                        IF fb_json.HasMember(json_FeederConfig, 'InFilterDelay') THEN
                            json_value := fb_json.FindMember(json_FeederConfig, 'InFilterDelay');
                            PERS.recipeList[i + 0].st110.FeederConfig.InFilterDelay
                                := TO_DINT(fb_json.GetInt(json_value));
                        END_IF

                        IF fb_json.HasMember(json_FeederConfig, 'StartDelay') THEN
                            json_value := fb_json.FindMember(json_FeederConfig, 'StartDelay');
                            PERS.recipeList[i + 0].st110.FeederConfig.StartDelay
                                := TO_DINT(fb_json.GetInt(json_value));
                        END_IF

                        IF fb_json.HasMember(json_FeederConfig, 'StopDelay') THEN
                            json_value := fb_json.FindMember(json_FeederConfig, 'StopDelay');
                            PERS.recipeList[i + 0].st110.FeederConfig.StopDelay
                                := TO_DINT(fb_json.GetInt(json_value));
                        END_IF

                        IF fb_json.HasMember(json_FeederConfig, 'EmptyDelay') THEN
                            json_value := fb_json.FindMember(json_FeederConfig, 'EmptyDelay');
                            PERS.recipeList[i + 0].st110.FeederConfig.EmptyDelay
                                := TO_DINT(fb_json.GetInt(json_value));
                        END_IF
                    END_IF
                END_IF

                IF fb_json.HasMember(json_i, 'st115') THEN
                    json_st115 := fb_json.FindMember(json_i, 'st115');

                    IF fb_json.HasMember(json_st115, 'xUseVerLeft') THEN
                        json_value                               := fb_json.FindMember(json_st115, 'xUseVerLeft');
                        PERS.recipeList[i + 0].st115.xUseVerLeft := TO_BOOL(fb_json.GetBool(json_value));
                    END_IF

                    IF fb_json.HasMember(json_st115, 'xUseVerRight') THEN
                        json_value                                := fb_json.FindMember(json_st115, 'xUseVerRight');
                        PERS.recipeList[i + 0].st115.xUseVerRight := TO_BOOL(fb_json.GetBool(json_value));
                    END_IF

                    IF fb_json.HasMember(json_st115, 'FeederConfig') THEN
                        json_FeederConfig := fb_json.FindMember(json_st115, 'FeederConfig');

                        IF fb_json.HasMember(json_FeederConfig, 'InFilterDelay') THEN
                            json_value := fb_json.FindMember(json_FeederConfig, 'InFilterDelay');
                            PERS.recipeList[i + 0].st115.FeederConfig.InFilterDelay
                                := TO_DINT(fb_json.GetInt(json_value));
                        END_IF

                        IF fb_json.HasMember(json_FeederConfig, 'StartDelay') THEN
                            json_value := fb_json.FindMember(json_FeederConfig, 'StartDelay');
                            PERS.recipeList[i + 0].st115.FeederConfig.StartDelay
                                := TO_DINT(fb_json.GetInt(json_value));
                        END_IF

                        IF fb_json.HasMember(json_FeederConfig, 'StopDelay') THEN
                            json_value := fb_json.FindMember(json_FeederConfig, 'StopDelay');
                            PERS.recipeList[i + 0].st115.FeederConfig.StopDelay
                                := TO_DINT(fb_json.GetInt(json_value));
                        END_IF

                        IF fb_json.HasMember(json_FeederConfig, 'EmptyDelay') THEN
                            json_value := fb_json.FindMember(json_FeederConfig, 'EmptyDelay');
                            PERS.recipeList[i + 0].st115.FeederConfig.EmptyDelay
                                := TO_DINT(fb_json.GetInt(json_value));
                        END_IF
                    END_IF
                END_IF

                IF fb_json.HasMember(json_i, 'st120') THEN
                    json_st120 := fb_json.FindMember(json_i, 'st120');

                    IF fb_json.HasMember(json_st120, 'xUseVerLeft') THEN
                        json_value                               := fb_json.FindMember(json_st120, 'xUseVerLeft');
                        PERS.recipeList[i + 0].st120.xUseVerLeft := TO_BOOL(fb_json.GetBool(json_value));
                    END_IF

                    IF fb_json.HasMember(json_st120, 'xUseVerRight') THEN
                        json_value                                := fb_json.FindMember(json_st120, 'xUseVerRight');
                        PERS.recipeList[i + 0].st120.xUseVerRight := TO_BOOL(fb_json.GetBool(json_value));
                    END_IF

                    IF fb_json.HasMember(json_st120, 'FeederConfigLeft') THEN
                        json_FeederConfigLeft := fb_json.FindMember(json_st120, 'FeederConfigLeft');

                        IF fb_json.HasMember(json_FeederConfigLeft, 'InFilterDelay') THEN
                            json_value := fb_json.FindMember(json_FeederConfigLeft, 'InFilterDelay');
                            PERS.recipeList[i + 0].st120.FeederConfigLeft.InFilterDelay
                                := TO_DINT(fb_json.GetInt(json_value));
                        END_IF

                        IF fb_json.HasMember(json_FeederConfigLeft, 'StartDelay') THEN
                            json_value := fb_json.FindMember(json_FeederConfigLeft, 'StartDelay');
                            PERS.recipeList[i + 0].st120.FeederConfigLeft.StartDelay
                                := TO_DINT(fb_json.GetInt(json_value));
                        END_IF

                        IF fb_json.HasMember(json_FeederConfigLeft, 'StopDelay') THEN
                            json_value := fb_json.FindMember(json_FeederConfigLeft, 'StopDelay');
                            PERS.recipeList[i + 0].st120.FeederConfigLeft.StopDelay
                                := TO_DINT(fb_json.GetInt(json_value));
                        END_IF

                        IF fb_json.HasMember(json_FeederConfigLeft, 'EmptyDelay') THEN
                            json_value := fb_json.FindMember(json_FeederConfigLeft, 'EmptyDelay');
                            PERS.recipeList[i + 0].st120.FeederConfigLeft.EmptyDelay
                                := TO_DINT(fb_json.GetInt(json_value));
                        END_IF
                    END_IF

                    IF fb_json.HasMember(json_st120, 'FeederConfigRight') THEN
                        json_FeederConfigRight := fb_json.FindMember(json_st120, 'FeederConfigRight');

                        IF fb_json.HasMember(json_FeederConfigRight, 'InFilterDelay') THEN
                            json_value := fb_json.FindMember(json_FeederConfigRight, 'InFilterDelay');
                            PERS.recipeList[i + 0].st120.FeederConfigRight.InFilterDelay
                                := TO_DINT(fb_json.GetInt(json_value));
                        END_IF

                        IF fb_json.HasMember(json_FeederConfigRight, 'StartDelay') THEN
                            json_value := fb_json.FindMember(json_FeederConfigRight, 'StartDelay');
                            PERS.recipeList[i + 0].st120.FeederConfigRight.StartDelay
                                := TO_DINT(fb_json.GetInt(json_value));
                        END_IF

                        IF fb_json.HasMember(json_FeederConfigRight, 'StopDelay') THEN
                            json_value := fb_json.FindMember(json_FeederConfigRight, 'StopDelay');
                            PERS.recipeList[i + 0].st120.FeederConfigRight.StopDelay
                                := TO_DINT(fb_json.GetInt(json_value));
                        END_IF

                        IF fb_json.HasMember(json_FeederConfigRight, 'EmptyDelay') THEN
                            json_value := fb_json.FindMember(json_FeederConfigRight, 'EmptyDelay');
                            PERS.recipeList[i + 0].st120.FeederConfigRight.EmptyDelay
                                := TO_DINT(fb_json.GetInt(json_value));
                        END_IF
                    END_IF
                END_IF

                IF fb_json.HasMember(json_i, 'st125') THEN
                    json_st125 := fb_json.FindMember(json_i, 'st125');

                    IF fb_json.HasMember(json_st125, 'xUseVerLeft') THEN
                        json_value := fb_json.FindMember(json_st125, 'xUseVerLeft');
                        PERS.recipeList[i + 0].st125.xUseVerLeft
                            := TO_BOOL(fb_json.GetBool(json_value));
                    END_IF

                    IF fb_json.HasMember(json_st125, 'xUseVerRight') THEN
                        json_value := fb_json.FindMember(json_st125, 'xUseVerRight');
                        PERS.recipeList[i + 0].st125.xUseVerRight
                            := TO_BOOL(fb_json.GetBool(json_value));
                    END_IF

                    IF fb_json.HasMember(json_st125, 'FeederConfig') THEN
                        json_FeederConfig := fb_json.FindMember(json_st125, 'FeederConfig');

                        IF fb_json.HasMember(json_FeederConfig, 'InFilterDelay') THEN
                            json_value := fb_json.FindMember(json_FeederConfig, 'InFilterDelay');
                            PERS.recipeList[i + 0].st125.FeederConfig.InFilterDelay
                                := TO_DINT(fb_json.GetInt(json_value));
                        END_IF

                        IF fb_json.HasMember(json_FeederConfig, 'StartDelay') THEN
                            json_value := fb_json.FindMember(json_FeederConfig, 'StartDelay');
                            PERS.recipeList[i + 0].st125.FeederConfig.StartDelay
                                := TO_DINT(fb_json.GetInt(json_value));
                        END_IF

                        IF fb_json.HasMember(json_FeederConfig, 'StopDelay') THEN
                            json_value := fb_json.FindMember(json_FeederConfig, 'StopDelay');
                            PERS.recipeList[i + 0].st125.FeederConfig.StopDelay
                                := TO_DINT(fb_json.GetInt(json_value));
                        END_IF

                        IF fb_json.HasMember(json_FeederConfig, 'EmptyDelay') THEN
                            json_value := fb_json.FindMember(json_FeederConfig, 'EmptyDelay');
                            PERS.recipeList[i + 0].st125.FeederConfig.EmptyDelay
                                := TO_DINT(fb_json.GetInt(json_value));
                        END_IF
                    END_IF
                END_IF

                IF fb_json.HasMember(json_i, 'st145') THEN
                    json_st145 := fb_json.FindMember(json_i, 'st145');

                    IF fb_json.HasMember(json_st145, 'xUseVerLeft') THEN
                        json_value := fb_json.FindMember(json_st145, 'xUseVerLeft');
                        PERS.recipeList[i + 0].st145.xUseVerLeft
                            := TO_BOOL(fb_json.GetBool(json_value));
                    END_IF

                    IF fb_json.HasMember(json_st145, 'xUseVerRight') THEN
                        json_value := fb_json.FindMember(json_st145, 'xUseVerRight');
                        PERS.recipeList[i + 0].st145.xUseVerRight
                            := TO_BOOL(fb_json.GetBool(json_value));
                    END_IF

                    IF fb_json.HasMember(json_st145, 'FeederConfig') THEN
                        json_FeederConfig := fb_json.FindMember(json_st145, 'FeederConfig');

                        IF fb_json.HasMember(json_FeederConfig, 'InFilterDelay') THEN
                            json_value := fb_json.FindMember(json_FeederConfig, 'InFilterDelay');
                            PERS.recipeList[i + 0].st145.FeederConfig.InFilterDelay
                                := TO_DINT(fb_json.GetInt(json_value));
                        END_IF

                        IF fb_json.HasMember(json_FeederConfig, 'StartDelay') THEN
                            json_value := fb_json.FindMember(json_FeederConfig, 'StartDelay');
                            PERS.recipeList[i + 0].st145.FeederConfig.StartDelay
                                := TO_DINT(fb_json.GetInt(json_value));
                        END_IF

                        IF fb_json.HasMember(json_FeederConfig, 'StopDelay') THEN
                            json_value := fb_json.FindMember(json_FeederConfig, 'StopDelay');
                            PERS.recipeList[i + 0].st145.FeederConfig.StopDelay
                                := TO_DINT(fb_json.GetInt(json_value));
                        END_IF

                        IF fb_json.HasMember(json_FeederConfig, 'EmptyDelay') THEN
                            json_value := fb_json.FindMember(json_FeederConfig, 'EmptyDelay');
                            PERS.recipeList[i + 0].st145.FeederConfig.EmptyDelay
                                := TO_DINT(fb_json.GetInt(json_value));
                        END_IF
                    END_IF
                END_IF
            END_IF

            IF fb_json.HasMember(json_i, 'st180') THEN
                json_st180 := fb_json.FindMember(json_i, 'st180');

                IF fb_json.HasMember(json_st180, 'xUseVerLeft') THEN
                    json_value                               := fb_json.FindMember(json_st180, 'xUseVerLeft');
                    PERS.recipeList[i + 0].st180.xUseVerLeft := TO_BOOL(fb_json.GetBool(json_value));
                END_IF

                IF fb_json.HasMember(json_st180, 'xUseVerRight') THEN
                    json_value                                := fb_json.FindMember(json_st180, 'xUseVerRight');
                    PERS.recipeList[i + 0].st180.xUseVerRight := TO_BOOL(fb_json.GetBool(json_value));
                END_IF
            END_IF
        END_FOR
    END_IF
END_IF

IF fb_json.HasMember(json_head, 'iRecipeCurrent') THEN
    json_value          := fb_json.FindMember(json_head, 'iRecipeCurrent');
    PERS.iRecipeCurrent := TO_INT(fb_json.GetInt(json_value));
END_IF

END_FUNCTION

// ---- POUs/20_AUTO/FileMan/LoadFromMemory.TcPOU
FUNCTION LoadFromMemory : BOOL
VAR_INPUT
    sData : REFERENCE TO STRING(2000);
END_VAR
VAR
    fbJson     : FB_JsonSaxReader;
    pJsonParse : FB_ReadJSON;
    //pJsonParse : FB_ReadRecipeJson;

    i : int;
END_VAR

// pJsonParse.myArrayInput1 REF= PERS.iStationTimeDef1;
// pJsonParse.myArrayInput2 REF= PERS.iStationTimeDef2;
fbJson.Parse(sJson := sData, ipHdl := pJsonParse);

END_FUNCTION

// ---- POUs/20_AUTO/FileMan/SaveInMemory.TcPOU
FUNCTION SaveInMemory : BOOL
VAR_INPUT
    sData : REFERENCE TO STRING(2000);
END_VAR
VAR
    fbJson     : FB_JsonSaxWriter;
    i          : int;
END_VAR

fbJson.ResetDocument();
// global object
fbJson.StartObject();
fbJson.AddKey('StationTimeArray');

// array1
fbJson.StartObject();
fbJson.AddKey('StationTime1');
fbJson.StartArray();

FOR i := 1 TO CONST.STATION_NUMBER BY 1 DO
    fbJson.AddDint(PERS.iStationTimeDef1[i]);
END_FOR

fbJson.EndArray();

// array2
fbJson.AddKey('StationTime2');
fbJson.StartArray();

FOR i := 1 TO CONST.STATION_NUMBER BY 1 DO
    fbJson.AddDint(PERS.iStationTimeDef2[i]);
END_FOR


fbJson.EndArray();
fbJson.EndObject();

fbJson.EndObject();
// end global object

// end of file
sData := fbJson.GetDocument();

fbJson.ResetDocument();

END_FUNCTION

// ---- POUs/20_AUTO/ST100/FB_ABL_LASER.TcPOU
FUNCTION_BLOCK FB_ABL_LASER
(****************************************************************************************)
(*	TITEL				Bezeichnung Ablauf	    										*)
(*	Status				ungetestet                         								*)
(*  Version:			1.0																*)
(*	Beschrieb:			Ablaufbeschreibung												*)
(*																						*)
(*	Steps:																				*)
(*		RESET:=0		Reset der Station												*)
(* 		INIT:=100		Initialisieren													*)
(*		... 			...																*)
(*		READY:=999		Initialisiert, Bereit für Start									*)
(*		START:=1000		Start Zyklisch 													*)
(*		... 			...																*)
(*		DONE:=8000		Letzer Schritt													*)
(*		ERROR:=9000		ALARM/Fehler													*)
(* 	09.09.2019/Dj																		*)
(***********************************Revisionen*******************************************)
(*	dd.mm.yyyy   KZ    x.y			Beschrieb											*)
(****************************************************************************************)

VAR_INPUT
    xIN_Reset       : BOOL;          // Schrittkette zurücksetzen 
    xIN_Init        : BOOL;          // Initialisieren
    xIN_Quit        : BOOL;          // Fehler quittieren 
    xIN_Start       : BOOL;          // Startbefehl
    xIN_Sperre      : BOOL;          // FB Sperren 
    xIN_NextStep    : BOOL;          // Nächsten Schritt ausführen 
    xIN_AlarmAktiv  : BOOL;          // Anlage hat Alarm
    xIN_DryCycle    : BOOL;          // Fahren ohne Teile
    xIN_RestartCYCL : BOOL;          // Zyklus erneut starten im STEP, END, LEERFAHREN
    enIN_State      : enState;       // Status Anlage
    tIN_Timeout     : TIME := T#10s; // Timout

    pxFG_Freigabe : POINTER TO BOOL; //Freigabe von Station

    // Application specific
    iProcessTimeMili1 : UDINT := 5000; // user defined station duration, in milisecond
    iProcessTimeMili2 : UDINT := 5000; // user defined station duration, in milisecond
    Mover            : REFERENCE TO FB_Mover;
    //xIN_MoverInPos  : BOOL;          // Set this flag when a mover is in position and ready to be handled
END_VAR
VAR_OUTPUT
    (* standart Ausgänge *)
    xOUT_ErrFlag     : BOOL;   // Error Flag 
    xOUT_Busy        : BOOL;   // Baustein befindet sich im Ablauf 
    xOUT_Done        : BOOL;   // Baustein hat den Ablauf beendet 		
    xOUT_Ready       : BOOL;   // Ready to begin, should be the same state as done	
    xOUT_Timeout     : BOOL;   // Timeout FB 
    xOUT_InitDone    : BOOL;   // initialisierung fertig
    xOUT_Wait        : BOOL;   // Wartet auf Bedingung
    iOUT_Step        : INT;    // Aktueller Schritt 
    sOUT_Step        : STRING; // Aktueller Schritt but in string format
    bOUT_Error       : BYTE;   // Fehlernummer

    xOUT_MoverFree   : BOOL;   // The mover is free to move
    //xOUT_MoverNeeded : BOOL;   // A mover is needed by this station to continue its process
    iOUT_ProcessCompletion : INT; //process completion, express in % (0-100)
END_VAR
VAR
    (* Standard *)
    (* Schritt *)
    iLastStep : INT; // Merker letzter Schritt 
    iPreStep  : INT; // Schritt zurück nach Alarm 
    iAktStep  : INT; // aktueller Schritt

    // Trigger Starten 
    rtSTART : R_TRIG;
    // Timer TimeOut 
    TON_Timeout : TON;

    (* Bausteine *)

    (* Spezial *)
    iStartProcessTimeMili : UDINT; // start of the processing time, accurate at 100ns 
	
	_bBewegung : BOOL;
	_bBewegungDist : INT := 20;

END_VAR
VAR CONSTANT
END_VAR

(*******************************************************************)
(* Trigger  *)
(*******************************************************************)
(* Zurücksetzen *)
IF xIN_RESET THEN
    iPreStep  := ST100_Laser_e.RESET;
    iOUT_Step := ST100_Laser_e.RESET;
END_IF;

(* Error Quittieren *)
IF (bOUT_Error <> 0) AND xIN_Quit THEN
    xOUT_ErrFlag := FALSE;
    bOUT_Error   := 0;
    iOUT_Step    := iPreStep;
END_IF;

(*******************************************************************)
(* Timer *)
(*******************************************************************)
TON_Timeout(IN := xIN_NextStep AND (iLastStep = iOUT_Step) (*todo FG *) ,
            PT := tIN_Timeout);

(*******************************************************************)
(* Bausteine *)
(*******************************************************************)

(*******************************************************************)
(* OUTPUTS *)
(*******************************************************************)
// Error Flag 
xOUT_ErrFlag := (bOUT_Error <> 0);
// Baustein befindet sich im Ablauf 
xOUT_Busy := (iOUT_Step > ST100_Laser_e.READY) AND (iOUT_Step < ST100_Laser_e.DONE);
// Baustein hat den Ablauf beendet
xOUT_Done := (iOUT_Step = ST100_Laser_e.DONE);
// Process ready
xOUT_Ready := (iOUT_Step = ST100_Laser_e.READY);
// Timeout FB 				 		
xOUT_Timeout := TON_Timeout.Q;
// Itialisierung fertig			
xOUT_InitDone := (iOUT_Step = ST100_Laser_e.READY);
// Aktueller Schritt			
iOUT_Step := iOUT_Step; //Im Ablauf gesetzt		
sOUT_Step := TO_STRING(iOUT_Step);
//Fehlernummer	 
bOUT_Error := bOUT_Error; //Im Ablauf/FB gesetzt	
(* Warte (alle Schritte wo auf FG oder Teile gewartet wird) *)
xOUT_Wait := (iOUT_Step = ST100_Laser_e.DONE);

xOUT_MoverFree := iOUT_Step = ST100_Laser_e.waitOnMover;

iOUT_ProcessCompletion := F_GetPercent(iAktStep,
                                       ST100_Laser_e.START,
                                       ST100_Laser_e.DONE,
                                       ST100_Laser_e.proceedOperation_1,
                                       ST100_Laser_e.proceedOperation_2,
                                       iStartProcessTimeMili,
                                       TO_DINT(iProcessTimeMili1),
                                       TO_DINT(iProcessTimeMili2));

(*******************************************************************)
(* Ablauf *)
(*******************************************************************)

(* Sperren *)
IF xIN_Sperre THEN
    iPreStep  := ST100_Laser_e.RESET;
    iOUT_Step := ST100_Laser_e.RESET;
    RETURN;
END_IF;

(* Schritt Merker *)
IF iAktStep <> iOUT_Step THEN
    iLastStep := iAktStep;
    iAktStep  := iOUT_Step;
END_IF

(* START *)
rtSTART(CLK := xIN_Start);

(*******************************************************************)
(* Schrittkette  *)
(*******************************************************************)
CASE iOUT_Step OF

(***** RESET *****)
ST100_Laser_e.RESET: (* Schritt 0-99 *)
    //Initialisierungen
    //Start Init Ablauf
    IF xIN_Init THEN
        iOUT_Step := ST100_Laser_e.INIT;
        //Start Manu Ablauf
    ELSIF enIN_State = StateMANU AND xIN_NextStep THEN
        iOUT_Step := ST100_Laser_e.INIT;
    END_IF;

(***** INIT *****)
ST100_Laser_e.INIT: (* Grundstellung ? *)
    IF TRUE THEN
        iOUT_Step := ST100_Laser_e.READY;
    ELSE
        iOUT_Step := ST100_Laser_e.INIT;
    END_IF;

(***** READY / INIT DONE *****)
ST100_Laser_e.READY:  (* Start AUTO,END,LEER,STEP *)
    IF xIN_Start THEN //IF rtSTART.Q THEN
        iOUT_Step := ST100_Laser_e.START;
    END_IF

(***** START  ZYKLISCH *****)
ST100_Laser_e.START: (*  *)
    IF xIN_NextStep AND pxFG_Freigabe^ THEN
        iOUT_Step             := ST100_Laser_e.waitOnMover;
        iStartProcessTimeMili := GetTick();
    END_IF;

ST100_Laser_e.waitOnMover: (*  *)
    IF xIN_NextStep AND __ISVALIDREF(Mover) THEN
        iStartProcessTimeMili := GetTick();
        iOUT_Step             := ST100_Laser_e.proceedOperation_1;
    END_IF;

ST100_Laser_e.proceedOperation_1: (*  *)
    IF xIN_NextStep AND (GetTick() - iStartProcessTimeMili) >= (iProcessTimeMili1) THEN
        iStartProcessTimeMili := GetTick();
        iOUT_Step             := ST100_Laser_e.proceedOperation_2;
        _bBewegung            := FALSE;
    END_IF

ST100_Laser_e.move_mover_to_next_piece:
    IF __ISVALIDREF(Mover) THEN
        IF Mover.MoverAxis.RelMoveTo(120.0).isInPos THEN
            iOUT_Step := ST100_Laser_e.proceedOperation_2;
        END_IF
    END_IF;

ST100_Laser_e.proceedOperation_2: (*  *)
    IF xIN_NextStep AND (GetTick() - iStartProcessTimeMili) >= (iProcessTimeMili2) THEN
        iOUT_Step := ST100_Laser_e.SYNC_MOVER_LEAVE;
    END_IF;

ST100_Laser_e.SYNC_MOVER_LEAVE:
    // The mover needs to be taken by MoverMan
    IF NOT __ISVALIDREF(Mover) THEN
        iOUT_Step := ST100_Unload_e.DONE;
    END_IF

(***** DONE *****)
ST100_Laser_e.DONE: (* Letzter Schritt  *)
    IF NOT xIN_AlarmAktiv THEN
        //AUTO
        IF (enIN_State = StateAUTO) AND xIN_RestartCYCL THEN
            iOUT_Step := ST100_Laser_e.START;
            //STEP / END / LEERFAHREN restart
        ELSIF (enIN_State < StateAUTO) AND (enIN_State >= enState.StateSTEP) AND xIN_RestartCYCL THEN
            iOUT_Step := ST100_Laser_e.START;
            //STEP / END / LEERFAHREN fertig
        ELSIF (enIN_State = StateREADY) THEN
            iOUT_Step := ST100_Laser_e.READY;
        END_IF;
    END_IF;

(************ ERROR *************)
ST100_Laser_e.ERROR: (* ERROR *) ;

END_CASE;

END_FUNCTION_BLOCK

// ---- POUs/20_AUTO/ST100/FB_AUT_LASER.TcPOU
FUNCTION_BLOCK FB_AUT_LASER EXTENDS FB_AUT_ABSTRACT IMPLEMENTS ISimuMoverTimers
    (****************************************************************************)
    (*	POU_AUT_zxx			Bausteinaufrufe Station	zxx							*)
    (*	Status				ungetestet											*)
    (*  Version:			1.0													*)
    (*	Beschrieb:																*)
    (*																			*)
    (*	Abläufe:			FB_ABLzxxA		Hauptablauf							*)
    (*																			*)
    (*																			*)
    (* 	25.09.2019/Dj															*)
    (****************************************************************************)
    (*	dd.mm.yyyy   KZ    x.y			Beschrieb								*)
    (****************************************************************************)
VAR_INPUT
    (* spezifische Eingänge *)

END_VAR
VAR_OUTPUT
    (* spezifische Ausgänge *)

END_VAR
VAR
    (* Bausteine *)
    _FB_ABL_100A : FB_ABL_LASER;
END_VAR

(*******************************************************************)
(* Timer *)
(*******************************************************************)

(*******************************************************************)
(* Flanken / Merker *)
(*******************************************************************)
//MANU CYCLE
IF (enIN_State = StateMANU) AND xIN_ManuCycle THEN
    xManuCycle := TRUE;
END_IF;

IF (enIN_State <> StateMANU) OR xOUT_Done THEN
    xManuCycle := FALSE;
END_IF

//NEXT STEP
xNextStep := (enIN_State > StateSTEP) OR
             ((enIN_State = StateSTEP) AND xIN_Step) OR
             ((enIN_State = StateMANU) AND xManuCycle);

//RESET
xReset := (enIN_State < StateREADY) AND (enIN_State <> StateINIT) AND NOT xManuCycle;

(*******************************************************************)
(* Bausteinaufrufe Abläufe *)
(*******************************************************************)

_FB_ABL_100A(xIN_Reset    := xReset,
             xIN_Init     := xIN_Init,
             xIN_Quit     := xIN_Quit,
             xIN_Start    := enIN_State = enState.StateAUTO, //AND _FB_ABL_100A.xOUT_Done AND _FB_ABL_100A.xOUT_Ready,
             xIN_Sperre   := NOT xIN_On,
             xIN_NextStep := xNextStep,
             xIN_AlarmAktiv
                 := xIN_AlarmAktiv,
             xIN_DryCycle    := xIN_DryCycle,
             xIN_RestartCYCL := enIN_State = enState.StateAUTO, // only restart when the mover has move out
             enIN_State      := enIN_State,
             tIN_Timeout     := tIN_Timeout,
             pxFG_Freigabe   := ADR(xRelease),
             Mover           := THIS^.Mover,
             xOUT_ErrFlag    =>,
             xOUT_Busy       =>,
             xOUT_Done       =>,
             xOUT_Timeout    =>,
             xOUT_InitDone   =>,
             xOUT_Wait       =>,
             iOUT_Step       =>,
             bOUT_Error      =>);

(*******************************************************************)
(* Mover reset flags *)
(*******************************************************************)

(*******************************************************************)
(* OUTPUT *)
(*******************************************************************)
xOUT_InitDone := _FB_ABL_100A.xOUT_InitDone;
xOUT_Ready    := xOUT_InitDone;
xOUT_Done     := _FB_ABL_100A.xOUT_Done;
xOUT_ErrFlag  := _FB_ABL_100A.xOUT_ErrFlag;
xOUT_Wait     := _FB_ABL_100A.xOUT_Wait;
xOUT_AlarmST  := xOUT_ErrFlag;

(*******************************************************************)
(* Bausteinaufruf Error Station *)
(*******************************************************************)
// POU_ERR_VORLAGE(xIN_QUIT:=xIN_Quit , pstrArIN_ALARM:=ADR(HMI.strArALARM[1]));

METHOD GiveMover : IProcessSampleMover
VAR_INPUT
	mover : REFERENCE TO FB_Mover;
END_VAR
IF __ISVALIDREF(mover) THEN
    THIS^.Mover                       REF= mover;
END_IF
END_METHOD

(* % of completion of the process *)
PROPERTY iCompletionPC : INT
GET
iCompletionPC := THIS^._FB_ABL_100A.iOUT_ProcessCompletion;
END_GET
END_PROPERTY

(* Process time, expressed in milisecond *)
PROPERTY iProcessTimeMili_1 : DINT
GET
iProcessTimeMili_1 := TO_DINT(this^._FB_ABL_100A.iProcessTimeMili1);
END_GET
SET
THIS^._FB_ABL_100A.iProcessTimeMili1 := TO_UDINT(iProcessTimeMili_1);
END_SET
END_PROPERTY

(* Process time, expressed in milisecond *)
PROPERTY iProcessTimeMili_2 : DINT
GET
iProcessTimeMili_2 := TO_DINT(this^._FB_ABL_100A.iProcessTimeMili2);
END_GET
SET
THIS^._FB_ABL_100A.iProcessTimeMili2 := TO_UDINT(iProcessTimeMili_2);
END_SET
END_PROPERTY

PROPERTY ProcessExecution : ProcessExecution_e
GET
ProcessExecution := THIS^._ProcessExecution;
END_GET
SET
THIS^._ProcessExecution := ProcessExecution;
END_SET
END_PROPERTY

METHOD TakeMover : IProcessSampleMover
VAR_INPUT
END_VAR
THIS^.Mover REF= 0;
END_METHOD

PROPERTY xBusy : BOOL
GET
xBusy := This^._FB_ABL_100A.xOUT_Busy;
END_GET
SET
END_SET
END_PROPERTY

PROPERTY xDone : BOOL
GET
xDone := THIS^._FB_ABL_100A.xOUT_Ready OR THIS^._FB_ABL_100A.xOUT_Done;
END_GET
END_PROPERTY

PROPERTY xMoverPathFree : BOOL
GET
xMoverPathFree := THIS^._FB_ABL_100A.xOUT_MoverFree OR THIS^._FB_ABL_100A.xOUT_Ready OR THIS^._FB_ABL_100A.xOUT_Done;
END_GET
END_PROPERTY

PROPERTY xMoverShouldLeave : BOOL
GET
xMoverShouldLeave := THIS^._FB_ABL_100A.iOUT_Step = ST100_Modify_e.SYNC_MOVER_LEAVE;
END_GET
END_PROPERTY

END_FUNCTION_BLOCK

// ---- POUs/20_AUTO/ST100/FB_AUT_100.TcPOU
FUNCTION_BLOCK FB_AUT_100 EXTENDS FB_AUT_ABSTRACT IMPLEMENTS ISimuMoverTimers
    (****************************************************************************)
    (*	POU_AUT_zxx			Bausteinaufrufe Station	zxx							*)
    (*	Status				ungetestet											*)
    (*  Version:			1.0													*)
    (*	Beschrieb:																*)
    (*																			*)
    (*	Abläufe:			FB_ABLzxxA		Hauptablauf							*)
    (*																			*)
    (*																			*)
    (* 	25.09.2019/Dj															*)
    (****************************************************************************)
    (*	dd.mm.yyyy   KZ    x.y			Beschrieb								*)
    (****************************************************************************)
VAR_INPUT
    (* spezifische Eingänge *)

END_VAR
VAR_OUTPUT
    (* spezifische Ausgänge *)

END_VAR
VAR
    (* Bausteine *)
    _FB_ABL_100A : FB_ABL_LOAD;
END_VAR

(*******************************************************************)
(* Timer *)
(*******************************************************************)

(*******************************************************************)
(* Flanken / Merker *)
(*******************************************************************)
//MANU CYCLE
IF (enIN_State = StateMANU) AND xIN_ManuCycle THEN
    xManuCycle := TRUE;
END_IF;

IF (enIN_State <> StateMANU) OR xOUT_Done THEN
    xManuCycle := FALSE;
END_IF

//NEXT STEP
xNextStep := (enIN_State > StateSTEP) OR
             ((enIN_State = StateSTEP) AND xIN_Step) OR
             ((enIN_State = StateMANU) AND xManuCycle);

//RESET
xReset := (enIN_State < StateREADY) AND (enIN_State <> StateINIT) AND NOT xManuCycle;

(*******************************************************************)
(* Bausteinaufrufe Abläufe *)
(*******************************************************************)

_FB_ABL_100A(xIN_Reset    := xReset,
             xIN_Init     := xIN_Init,
             xIN_Quit     := xIN_Quit,
             xIN_Start    := enIN_State = enState.StateAUTO, //AND _FB_ABL_100A.xOUT_Done AND _FB_ABL_100A.xOUT_Ready,
             xIN_Sperre   := NOT xIN_On,
             xIN_NextStep := xNextStep,
             xIN_AlarmAktiv
                 := xIN_AlarmAktiv,
             xIN_DryCycle    := xIN_DryCycle,
             xIN_RestartCYCL := enIN_State = enState.StateAUTO, // only restart when the mover has move out
             enIN_State      := enIN_State,
             tIN_Timeout     := tIN_Timeout,
             pxFG_Freigabe   := ADR(xRelease),
             Mover           := THIS^.Mover,
             xOUT_ErrFlag    =>,
             xOUT_Busy       =>,
             xOUT_Done       =>,
             xOUT_Timeout    =>,
             xOUT_InitDone   =>,
             xOUT_Wait       =>,
             iOUT_Step       =>,
             bOUT_Error      =>);

(*******************************************************************)
(* Mover reset flags *)
(*******************************************************************)

(*******************************************************************)
(* OUTPUT *)
(*******************************************************************)
xOUT_InitDone := _FB_ABL_100A.xOUT_InitDone;
xOUT_Ready    := xOUT_InitDone;
xOUT_Done     := _FB_ABL_100A.xOUT_Done;
xOUT_ErrFlag  := _FB_ABL_100A.xOUT_ErrFlag;
xOUT_Wait     := _FB_ABL_100A.xOUT_Wait;
xOUT_AlarmST  := xOUT_ErrFlag;

(*******************************************************************)
(* Bausteinaufruf Error Station *)
(*******************************************************************)
// POU_ERR_VORLAGE(xIN_QUIT:=xIN_Quit , pstrArIN_ALARM:=ADR(HMI.strArALARM[1]));

METHOD GiveMover : IProcessSampleMover
VAR_INPUT
	mover : REFERENCE TO FB_Mover;
END_VAR
IF __ISVALIDREF(mover) THEN
    THIS^.Mover                       REF= mover;
END_IF
END_METHOD

(* % of completion of the process *)
PROPERTY iCompletionPC : INT
GET
iCompletionPC := THIS^._FB_ABL_100A.iOUT_ProcessCompletion;
END_GET
END_PROPERTY

(* Process time, expressed in milisecond *)
PROPERTY iProcessTimeMili_1 : DINT
GET
iProcessTimeMili_1 := TO_DINT(this^._FB_ABL_100A.iProcessTimeMili1);
END_GET
SET
THIS^._FB_ABL_100A.iProcessTimeMili1 := TO_UDINT(iProcessTimeMili_1);
END_SET
END_PROPERTY

(* Process time, expressed in milisecond *)
PROPERTY iProcessTimeMili_2 : DINT
GET
iProcessTimeMili_2 := TO_DINT(this^._FB_ABL_100A.iProcessTimeMili2);
END_GET
SET
THIS^._FB_ABL_100A.iProcessTimeMili2 := TO_UDINT(iProcessTimeMili_2);
END_SET
END_PROPERTY

PROPERTY ProcessExecution : ProcessExecution_e
GET
ProcessExecution := THIS^._ProcessExecution;
END_GET
SET
THIS^._ProcessExecution := ProcessExecution;
END_SET
END_PROPERTY

METHOD TakeMover : IProcessSampleMover
VAR_INPUT
END_VAR
THIS^.Mover REF= 0;
END_METHOD

PROPERTY xBusy : BOOL
GET
xBusy := This^._FB_ABL_100A.xOUT_Busy;
END_GET
SET
END_SET
END_PROPERTY

PROPERTY xDone : BOOL
GET
xDone := THIS^._FB_ABL_100A.xOUT_Ready OR THIS^._FB_ABL_100A.xOUT_Done;
END_GET
END_PROPERTY

PROPERTY xMoverPathFree : BOOL
GET
xMoverPathFree := THIS^._FB_ABL_100A.xOUT_MoverFree OR THIS^._FB_ABL_100A.xOUT_Ready OR THIS^._FB_ABL_100A.xOUT_Done;
END_GET
END_PROPERTY

PROPERTY xMoverShouldLeave : BOOL
GET
xMoverShouldLeave := THIS^._FB_ABL_100A.iOUT_Step = ST100_Load_e.SYNC_MOVER_LEAVE;
END_GET
END_PROPERTY

END_FUNCTION_BLOCK

// ---- POUs/20_AUTO/ST100/FB_ABL_LOAD.TcPOU
FUNCTION_BLOCK FB_ABL_LOAD
(****************************************************************************************)
(*	TITEL				Bezeichnung Ablauf	    										*)
(*	Status				ungetestet                         								*)
(*  Version:			1.0																*)
(*	Beschrieb:			Ablaufbeschreibung												*)
(*																						*)
(*	Steps:																				*)
(*		RESET:=0		Reset der Station												*)
(* 		INIT:=100		Initialisieren													*)
(*		... 			...																*)
(*		READY:=999		Initialisiert, Bereit für Start									*)
(*		START:=1000		Start Zyklisch 													*)
(*		... 			...																*)
(*		DONE:=8000		Letzer Schritt													*)
(*		ERROR:=9000		ALARM/Fehler													*)
(* 	09.09.2019/Dj																		*)
(***********************************Revisionen*******************************************)
(*	dd.mm.yyyy   KZ    x.y			Beschrieb											*)
(****************************************************************************************)

VAR_INPUT
    xIN_Reset       : BOOL;          // Schrittkette zurücksetzen 
    xIN_Init        : BOOL;          // Initialisieren
    xIN_Quit        : BOOL;          // Fehler quittieren 
    xIN_Start       : BOOL;          // Startbefehl
    xIN_Sperre      : BOOL;          // FB Sperren 
    xIN_NextStep    : BOOL;          // Nächsten Schritt ausführen 
    xIN_AlarmAktiv  : BOOL;          // Anlage hat Alarm
    xIN_DryCycle    : BOOL;          // Fahren ohne Teile
    xIN_RestartCYCL : BOOL;          // Zyklus erneut starten im STEP, END, LEERFAHREN
    enIN_State      : enState;       // Status Anlage
    tIN_Timeout     : TIME := T#10s; // Timout

    pxFG_Freigabe : POINTER TO BOOL; //Freigabe von Station

    // Application specific
    iProcessTimeMili1 : UDINT := 5000; // user defined station duration, in milisecond
    iProcessTimeMili2 : UDINT := 5000; // user defined station duration, in milisecond
    Mover            : REFERENCE TO FB_Mover;
    //xIN_MoverInPos  : BOOL;          // Set this flag when a mover is in position and ready to be handled
END_VAR
VAR_OUTPUT
    (* standart Ausgänge *)
    xOUT_ErrFlag     : BOOL;   // Error Flag 
    xOUT_Busy        : BOOL;   // Baustein befindet sich im Ablauf 
    xOUT_Done        : BOOL;   // Baustein hat den Ablauf beendet 		
    xOUT_Ready       : BOOL;   // Ready to begin, should be the same state as done	
    xOUT_Timeout     : BOOL;   // Timeout FB 
    xOUT_InitDone    : BOOL;   // initialisierung fertig
    xOUT_Wait        : BOOL;   // Wartet auf Bedingung
    iOUT_Step        : INT;    // Aktueller Schritt 
    sOUT_Step        : STRING; // Aktueller Schritt but in string format
    bOUT_Error       : BYTE;   // Fehlernummer

    iOUT_ProcessCompletion : INT; //process completion, express in % (0-100)
    xOUT_MoverFree   : BOOL;   // The mover is free to move
    //xOUT_MoverNeeded : BOOL;   // A mover is needed by this station to continue its process
END_VAR
VAR
    (* Standard *)
    (* Schritt *)
    iLastStep : INT; // Merker letzter Schritt 
    iPreStep  : INT; // Schritt zurück nach Alarm 
    iAktStep  : INT; // aktueller Schritt

    // Trigger Starten 
    rtSTART : R_TRIG;
    // Timer TimeOut 
    TON_Timeout : TON;

    (* Bausteine *)

    (* Spezial *)
    iStartProcessTimeMili : UDINT; // start of the processing time, accurate at 100ns 

END_VAR
VAR CONSTANT
END_VAR

(*******************************************************************)
(* Trigger  *)
(*******************************************************************)
(* Zurücksetzen *)
IF xIN_RESET THEN
    iPreStep  := ST100_Load_e.RESET;
    iOUT_Step := ST100_Load_e.RESET;
END_IF;

(* Error Quittieren *)
IF (bOUT_Error <> 0) AND xIN_Quit THEN
    xOUT_ErrFlag := FALSE;
    bOUT_Error   := 0;
    iOUT_Step    := iPreStep;
END_IF;

(*******************************************************************)
(* Timer *)
(*******************************************************************)
TON_Timeout(IN := xIN_NextStep AND (iLastStep = iOUT_Step) (*todo FG *) ,
            PT := tIN_Timeout);

(*******************************************************************)
(* Bausteine *)
(*******************************************************************)

(*******************************************************************)
(* OUTPUTS *)
(*******************************************************************)
// Error Flag 
xOUT_ErrFlag := (bOUT_Error <> 0);
// Baustein befindet sich im Ablauf 
xOUT_Busy := (iOUT_Step > ST100_Load_e.READY) AND (iOUT_Step < ST100_Load_e.DONE);
// Baustein hat den Ablauf beendet
xOUT_Done := (iOUT_Step = ST100_Load_e.DONE);
// Process ready
xOUT_Ready := (iOUT_Step = ST100_Load_e.READY);
// Timeout FB 				 		
xOUT_Timeout := TON_Timeout.Q;
// Itialisierung fertig			
xOUT_InitDone := (iOUT_Step = ST100_Load_e.READY);
// Aktueller Schritt			
iOUT_Step := iOUT_Step; //Im Ablauf gesetzt		
sOUT_Step := TO_STRING(iOUT_Step);
//Fehlernummer	 
bOUT_Error := bOUT_Error; //Im Ablauf/FB gesetzt	
(* Warte (alle Schritte wo auf FG oder Teile gewartet wird) *)
xOUT_Wait := (iOUT_Step = ST100_Load_e.DONE);

xOUT_MoverFree := iOUT_Step >= ST100_Load_e.MOVER_FREE_OP AND iOUT_Step < ST100_Load_e.MOVER_NEEDED_OP;

iOUT_ProcessCompletion := F_GetPercent(iAktStep,
                                       ST100_Load_e.START,
                                       ST100_Load_e.DONE,
                                       ST100_Load_e.proceedOperation_1,
                                       ST100_Load_e.proceedOperation_2,
                                       iStartProcessTimeMili,
                                       TO_DINT(iProcessTimeMili1),
                                       TO_DINT(iProcessTimeMili2));

(*******************************************************************)
(* Ablauf *)
(*******************************************************************)

(* Sperren *)
IF xIN_Sperre THEN
    iPreStep  := ST100_Load_e.RESET;
    iOUT_Step := ST100_Load_e.RESET;
    RETURN;
END_IF;

(* Schritt Merker *)
IF iAktStep <> iOUT_Step THEN
    iLastStep := iAktStep;
    iAktStep  := iOUT_Step;
END_IF

(* START *)
rtSTART(CLK := xIN_Start);

(*******************************************************************)
(* Schrittkette  *)
(*******************************************************************)
CASE iOUT_Step OF

(***** RESET *****)
ST100_Load_e.RESET: (* Schritt 0-99 *)
    //Initialisierungen
    //Start Init Ablauf
    IF xIN_Init THEN
        iOUT_Step := ST100_Load_e.INIT;
        //Start Manu Ablauf
    ELSIF enIN_State = StateMANU AND xIN_NextStep THEN
        iOUT_Step := ST100_Load_e.INIT;
    END_IF;

(***** INIT *****)
ST100_Load_e.INIT: (* Grundstellung ? *)
    IF TRUE THEN
        iOUT_Step := ST100_Load_e.READY;
    ELSE
        iOUT_Step := ST100_Load_e.INIT;
    END_IF;

(***** READY / INIT DONE *****)
ST100_Load_e.READY:   (* Start AUTO,END,LEER,STEP *)
    IF xIN_Start THEN //IF rtSTART.Q THEN
        iOUT_Step := ST100_Load_e.START;
    END_IF

(***** START  ZYKLISCH *****)
ST100_Load_e.START: (*  *)
    IF xIN_NextStep AND pxFG_Freigabe^ THEN
        iOUT_Step             := ST100_Load_e.proceedOperation_1;
        iStartProcessTimeMili := GetTick();
    END_IF;

ST100_Load_e.proceedOperation_1: (*  *)
    IF xIN_NextStep AND (GetTick() - iStartProcessTimeMili) >= (iProcessTimeMili1) THEN
        iOUT_Step := ST100_Load_e.waitOnMover;
    END_IF;

ST100_Load_e.waitOnMover: (*  *)
    IF xIN_NextStep AND __ISVALIDREF(Mover) THEN
        iStartProcessTimeMili := GetTick();
        iOUT_Step             := ST100_Load_e.proceedOperation_2;
    END_IF;

ST100_Load_e.proceedOperation_2: (*  *)
    IF xIN_NextStep AND (GetTick() - iStartProcessTimeMili) >= (iProcessTimeMili2) THEN
        iOUT_Step := ST100_Load_e.SYNC_MOVER_LEAVE;
    END_IF;

ST100_Load_e.SYNC_MOVER_LEAVE:
    // The mover needs to be taken by MoverMan
    IF NOT __ISVALIDREF(Mover) THEN
        iOUT_Step := ST100_Unload_e.DONE;
    END_IF

(***** DONE *****)
ST100_Load_e.DONE: (* Letzter Schritt  *)
    IF NOT xIN_AlarmAktiv THEN
        //AUTO
        IF (enIN_State = StateAUTO) AND xIN_RestartCYCL THEN
            iOUT_Step := ST100_Load_e.START;
            //STEP / END / LEERFAHREN restart
        ELSIF (enIN_State < StateAUTO) AND (enIN_State >= enState.StateSTEP) AND xIN_RestartCYCL THEN
            iOUT_Step := ST100_Load_e.START;
            //STEP / END / LEERFAHREN fertig
        ELSIF (enIN_State = StateREADY) THEN
            iOUT_Step := ST100_Load_e.READY;
        END_IF;
    END_IF;

(************ ERROR *************)
ST100_Load_e.ERROR: (* ERROR *) ;

END_CASE;

END_FUNCTION_BLOCK

// ---- POUs/20_AUTO/ST100/FB_ABL_UNLOAD.TcPOU
FUNCTION_BLOCK FB_ABL_UNLOAD
(****************************************************************************************)
(*	TITEL				Bezeichnung Ablauf	    										*)
(*	Status				ungetestet                         								*)
(*  Version:			1.0																*)
(*	Beschrieb:			Ablaufbeschreibung												*)
(*																						*)
(*	Steps:																				*)
(*		RESET:=0		Reset der Station												*)
(* 		INIT:=100		Initialisieren													*)
(*		... 			...																*)
(*		READY:=999		Initialisiert, Bereit für Start									*)
(*		START:=1000		Start Zyklisch 													*)
(*		... 			...																*)
(*		DONE:=8000		Letzer Schritt													*)
(*		ERROR:=9000		ALARM/Fehler													*)
(* 	09.09.2019/Dj																		*)
(***********************************Revisionen*******************************************)
(*	dd.mm.yyyy   KZ    x.y			Beschrieb											*)
(****************************************************************************************)

VAR_INPUT
    xIN_Reset       : BOOL;          // Schrittkette zurücksetzen 
    xIN_Init        : BOOL;          // Initialisieren
    xIN_Quit        : BOOL;          // Fehler quittieren 
    xIN_Start       : BOOL;          // Startbefehl
    xIN_Sperre      : BOOL;          // FB Sperren 
    xIN_NextStep    : BOOL;          // Nächsten Schritt ausführen 
    xIN_AlarmAktiv  : BOOL;          // Anlage hat Alarm
    xIN_DryCycle    : BOOL;          // Fahren ohne Teile
    xIN_RestartCYCL : BOOL;          // Zyklus erneut starten im STEP, END, LEERFAHREN
    enIN_State      : enState;       // Status Anlage
    tIN_Timeout     : TIME := T#10s; // Timout

    pxFG_Freigabe : POINTER TO BOOL; //Freigabe von Station

    // Application specific
    iProcessTimeMili : UDINT := 5000; // user defined station duration, in milisecond
    Mover            : REFERENCE TO FB_Mover;
    //xIN_MoverInPos  : BOOL;          // Set this flag when a mover is in position and ready to be handled
END_VAR
VAR_OUTPUT
    (* standart Ausgänge *)
    xOUT_ErrFlag     : BOOL;   // Error Flag 
    xOUT_Busy        : BOOL;   // Baustein befindet sich im Ablauf 
    xOUT_Done        : BOOL;   // Baustein hat den Ablauf beendet 		
    xOUT_Ready       : BOOL;   // Ready to begin, should be the same state as done	
    xOUT_Timeout     : BOOL;   // Timeout FB 
    xOUT_InitDone    : BOOL;   // initialisierung fertig
    xOUT_Wait        : BOOL;   // Wartet auf Bedingung
    xOUT_MoverFree   : BOOL;   // The mover is free to move
    //xOUT_MoverNeeded : BOOL;   // A mover is needed by this station to continue its process
    iOUT_Step        : INT;    // Aktueller Schritt 
    sOUT_Step        : STRING; // Aktueller Schritt but in string format
    bOUT_Error       : BYTE;   // Fehlernummer

    iOUT_ProcessCompletion : INT; //process completion, express in % (0-100)
END_VAR
VAR
    (* Standard *)
    (* Schritt *)
    iLastStep : INT; // Merker letzter Schritt 
    iPreStep  : INT; // Schritt zurück nach Alarm 
    iAktStep  : INT; // aktueller Schritt

    // Trigger Starten 
    rtSTART : R_TRIG;
    // Timer TimeOut 
    TON_Timeout : TON;

    (* Bausteine *)

    (* Spezial *)
    iStartProcessTimeMili : UDINT; // start of the processing time, accurate at 100ns 

END_VAR
VAR CONSTANT
END_VAR

(*******************************************************************)
(* Trigger  *)
(*******************************************************************)
(* Zurücksetzen *)
IF xIN_RESET THEN
    iPreStep  := ST100_Unload_e.RESET;
    iOUT_Step := ST100_Unload_e.RESET;
END_IF;

(* Error Quittieren *)
IF (bOUT_Error <> 0) AND xIN_Quit THEN
    xOUT_ErrFlag := FALSE;
    bOUT_Error   := 0;
    iOUT_Step    := iPreStep;
END_IF;

(*******************************************************************)
(* Timer *)
(*******************************************************************)
TON_Timeout(IN := xIN_NextStep AND (iLastStep = iOUT_Step) (*todo FG *) ,
            PT := tIN_Timeout);

(*******************************************************************)
(* Bausteine *)
(*******************************************************************)

(*******************************************************************)
(* OUTPUTS *)
(*******************************************************************)
// Error Flag 
xOUT_ErrFlag := (bOUT_Error <> 0);
// Baustein befindet sich im Ablauf 
xOUT_Busy := (iOUT_Step > ST100_Unload_e.READY) AND (iOUT_Step < ST100_Unload_e.DONE);
// Baustein hat den Ablauf beendet
xOUT_Done := (iOUT_Step = ST100_Unload_e.DONE);
// Process ready
xOUT_Ready := (iOUT_Step = ST100_Unload_e.READY);
// Timeout FB 				 		
xOUT_Timeout := TON_Timeout.Q;
// Itialisierung fertig			
xOUT_InitDone := (iOUT_Step = ST100_Unload_e.READY);
// Aktueller Schritt			
iOUT_Step := iOUT_Step; //Im Ablauf gesetzt		
sOUT_Step := TO_STRING(iOUT_Step);
//Fehlernummer	 
bOUT_Error := bOUT_Error; //Im Ablauf/FB gesetzt	
(* Warte (alle Schritte wo auf FG oder Teile gewartet wird) *)
xOUT_Wait := (iOUT_Step = ST100_Unload_e.DONE);

xOUT_MoverFree   := NOT (iOUT_Step >= ST100_Unload_e.MOVER_NEEDED_OP AND iOUT_Step < ST100_Unload_e.MOVER_FREE_OP);

IF iAktStep < ST100_Unload_e.START THEN
    iOUT_ProcessCompletion := 0;
ELSIF iAktStep > ST100_Unload_e.DONE THEN
    iOUT_ProcessCompletion :=
        getPercent(iPreStep, TO_INT(ST100_Unload_e.START), TO_INT(ST100_Unload_e.proceedOperation_2) + 1);
ELSIF ST100_Unload_e.DONE = iAktStep THEN
    iOUT_ProcessCompletion := 100;
ELSE
    // iOUT_ProcessCompletion := getPercent(iAktStep, TO_INT(ST100_Unload_e.START), TO_INT(ST100_Unload_e.releaseMover) + 1);
    IF iProcessTimeMili > 0 THEN
        IF iAktStep < ST100_Unload_e.proceedOperation_1 THEN
            iOUT_ProcessCompletion := 0;
        ELSIF iAktStep = ST100_Unload_e.proceedOperation_1 THEN
            iOUT_ProcessCompletion := TO_INT(((GetTick() - iStartProcessTimeMili) * 100) / iProcessTimeMili);
        ELSIF iAktStep = ST100_Unload_e.proceedOperation_2 THEN
            iOUT_ProcessCompletion := 50 + TO_INT(((GetTick() - iStartProcessTimeMili) * 100) / iProcessTimeMili);
        ELSE
            iOUT_ProcessCompletion := 50;
        END_IF
    ELSE
        iOUT_ProcessCompletion := 0;
    END_IF
END_IF

(*******************************************************************)
(* Ablauf *)
(*******************************************************************)

(* Sperren *)
IF xIN_Sperre THEN
    iPreStep  := ST100_Unload_e.RESET;
    iOUT_Step := ST100_Unload_e.RESET;
    RETURN;
END_IF;

(* Schritt Merker *)
IF iAktStep <> iOUT_Step THEN
    iLastStep := iAktStep;
    iAktStep  := iOUT_Step;
END_IF

(* START *)
rtSTART(CLK := xIN_Start);

(*******************************************************************)
(* Schrittkette  *)
(*******************************************************************)
CASE iOUT_Step OF

(***** RESET *****)
ST100_Unload_e.RESET: (* Schritt 0-99 *)
    //Initialisierungen
    //Start Init Ablauf
    IF xIN_Init THEN
        iOUT_Step := ST100_Unload_e.INIT;
        //Start Manu Ablauf
    ELSIF enIN_State = StateMANU AND xIN_NextStep THEN
        iOUT_Step := ST100_Unload_e.INIT;
    END_IF;

(***** INIT *****)
ST100_Unload_e.INIT: (* Grundstellung ? *)
    IF TRUE THEN
        iOUT_Step := ST100_Unload_e.READY;
    ELSE
        iOUT_Step := ST100_Unload_e.INIT;
    END_IF;

(***** READY / INIT DONE *****)
ST100_Unload_e.READY: (* Start AUTO,END,LEER,STEP *)
    IF xIN_Start THEN //IF rtSTART.Q THEN
        iOUT_Step := ST100_Unload_e.START;
    END_IF

(***** START  ZYKLISCH *****)
ST100_Unload_e.START: (*  *)
    IF xIN_NextStep AND pxFG_Freigabe^ THEN
        iOUT_Step := ST100_Unload_e.waitOnMover;
    END_IF;

ST100_Unload_e.waitOnMover: (*  *)
    IF xIN_NextStep AND __ISVALIDREF(Mover) THEN
        iStartProcessTimeMili := GetTick();
        iOUT_Step             := ST100_Unload_e.proceedOperation_1;
    END_IF;

ST100_Unload_e.proceedOperation_1: (*  *)
    IF xIN_NextStep AND (GetTick() - iStartProcessTimeMili) >= (iProcessTimeMili / 2) THEN
        iOUT_Step := ST100_Unload_e.SYNC_MOVER_LEAVE;
    END_IF;

ST100_Unload_e.SYNC_MOVER_LEAVE:
    // The mover needs to be taken by MoverMan
    IF NOT __ISVALIDREF(Mover) THEN
        iStartProcessTimeMili := GetTick();
        iOUT_Step             := ST100_Unload_e.proceedOperation_2;
    END_IF

ST100_Unload_e.proceedOperation_2: (*  *)
    IF xIN_NextStep AND (GetTick() - iStartProcessTimeMili) >= (iProcessTimeMili / 2) THEN
        iOUT_Step := ST100_Unload_e.DONE;
    END_IF;

(***** DONE *****)
ST100_Unload_e.DONE: (* Letzter Schritt  *)
    IF NOT xIN_AlarmAktiv THEN
        //AUTO
        IF (enIN_State = StateAUTO) AND xIN_RestartCYCL THEN
            iOUT_Step := ST100_Unload_e.START;
            //STEP / END / LEERFAHREN restart
        ELSIF (enIN_State < StateAUTO) AND (enIN_State >= enState.StateSTEP) AND xIN_RestartCYCL THEN
            iOUT_Step := ST100_Unload_e.START;
            //STEP / END / LEERFAHREN fertig
        ELSIF (enIN_State = StateREADY) THEN
            iOUT_Step := ST100_Unload_e.READY;
        END_IF;
    END_IF;

(************ ERROR *************)
ST100_Unload_e.ERROR: (* ERROR *) ;

END_CASE;

END_FUNCTION_BLOCK

// ---- POUs/20_AUTO/ST100/FB_AUT_LOAD.TcPOU
FUNCTION_BLOCK FB_AUT_LOAD EXTENDS FB_AUT_ABSTRACT IMPLEMENTS ISimuMoverTimers
    (****************************************************************************)
    (*	POU_AUT_zxx			Bausteinaufrufe Station	zxx							*)
    (*	Status				ungetestet											*)
    (*  Version:			1.0													*)
    (*	Beschrieb:																*)
    (*																			*)
    (*	Abläufe:			FB_ABLzxxA		Hauptablauf							*)
    (*																			*)
    (*																			*)
    (* 	25.09.2019/Dj															*)
    (****************************************************************************)
    (*	dd.mm.yyyy   KZ    x.y			Beschrieb								*)
    (****************************************************************************)
VAR_INPUT
    (* spezifische Eingänge *)

END_VAR
VAR_OUTPUT
    (* spezifische Ausgänge *)

END_VAR
VAR
    (* Bausteine *)
    _FB_ABL_100A : FB_ABL_LOAD;
END_VAR

(*******************************************************************)
(* Timer *)
(*******************************************************************)

(*******************************************************************)
(* Flanken / Merker *)
(*******************************************************************)
//MANU CYCLE
IF (enIN_State = StateMANU) AND xIN_ManuCycle THEN
    xManuCycle := TRUE;
END_IF;

IF (enIN_State <> StateMANU) OR xOUT_Done THEN
    xManuCycle := FALSE;
END_IF

//NEXT STEP
xNextStep := (enIN_State > StateSTEP) OR
             ((enIN_State = StateSTEP) AND xIN_Step) OR
             ((enIN_State = StateMANU) AND xManuCycle);

//RESET
xReset := (enIN_State < StateREADY) AND (enIN_State <> StateINIT) AND NOT xManuCycle;

(*******************************************************************)
(* Bausteinaufrufe Abläufe *)
(*******************************************************************)

_FB_ABL_100A(xIN_Reset    := xReset,
             xIN_Init     := xIN_Init,
             xIN_Quit     := xIN_Quit,
             xIN_Start    := enIN_State = enState.StateAUTO, //AND _FB_ABL_100A.xOUT_Done AND _FB_ABL_100A.xOUT_Ready,
             xIN_Sperre   := NOT xIN_On,
             xIN_NextStep := xNextStep,
             xIN_AlarmAktiv
                 := xIN_AlarmAktiv,
             xIN_DryCycle    := xIN_DryCycle,
             xIN_RestartCYCL := enIN_State = enState.StateAUTO, // only restart when the mover has move out
             enIN_State      := enIN_State,
             tIN_Timeout     := tIN_Timeout,
             pxFG_Freigabe   := ADR(xDummy),
             Mover           := THIS^.Mover,
             xOUT_ErrFlag    =>,
             xOUT_Busy       =>,
             xOUT_Done       =>,
             xOUT_Timeout    =>,
             xOUT_InitDone   =>,
             xOUT_Wait       =>,
             iOUT_Step       =>,
             bOUT_Error      =>);

(*******************************************************************)
(* Mover reset flags *)
(*******************************************************************)

(*******************************************************************)
(* OUTPUT *)
(*******************************************************************)
xOUT_InitDone := _FB_ABL_100A.xOUT_InitDone;
xOUT_Ready    := xOUT_InitDone;
xOUT_Done     := _FB_ABL_100A.xOUT_Done;
xOUT_ErrFlag  := _FB_ABL_100A.xOUT_ErrFlag;
xOUT_Wait     := _FB_ABL_100A.xOUT_Wait;
xOUT_AlarmST  := xOUT_ErrFlag;

(*******************************************************************)
(* Bausteinaufruf Error Station *)
(*******************************************************************)
// POU_ERR_VORLAGE(xIN_QUIT:=xIN_Quit , pstrArIN_ALARM:=ADR(HMI.strArALARM[1]));

METHOD GiveMover : IProcessSampleMover
VAR_INPUT
	mover : REFERENCE TO FB_Mover;
END_VAR
IF __ISVALIDREF(mover) THEN
    THIS^.Mover                       REF= mover;
END_IF
END_METHOD

(* % of completion of the process *)
PROPERTY iCompletionPC : INT
GET
iCompletionPC := THIS^._FB_ABL_100A.iOUT_ProcessCompletion;
END_GET
END_PROPERTY

(* Process time, expressed in milisecond *)
PROPERTY iProcessTimeMili_1 : DINT
GET
iProcessTimeMili_1 := TO_DINT(this^._FB_ABL_100A.iProcessTimeMili1);
END_GET
SET
THIS^._FB_ABL_100A.iProcessTimeMili1 := TO_UDINT(iProcessTimeMili_1);
END_SET
END_PROPERTY

(* Process time, expressed in milisecond *)
PROPERTY iProcessTimeMili_2 : DINT
GET
iProcessTimeMili_2 := TO_DINT(this^._FB_ABL_100A.iProcessTimeMili2);
END_GET
SET
THIS^._FB_ABL_100A.iProcessTimeMili2 := TO_UDINT(iProcessTimeMili_2);
END_SET
END_PROPERTY

PROPERTY ProcessExecution : ProcessExecution_e
GET
ProcessExecution := THIS^._ProcessExecution;
END_GET
SET
THIS^._ProcessExecution := ProcessExecution;
END_SET
END_PROPERTY

METHOD TakeMover : IProcessSampleMover
VAR_INPUT
END_VAR
THIS^.Mover REF= 0;
END_METHOD

PROPERTY xBusy : BOOL
GET
xBusy := This^._FB_ABL_100A.xOUT_Busy;
END_GET
SET
END_SET
END_PROPERTY

PROPERTY xDone : BOOL
GET
xDone := THIS^._FB_ABL_100A.xOUT_Ready OR THIS^._FB_ABL_100A.xOUT_Done;
END_GET
END_PROPERTY

PROPERTY xMoverPathFree : BOOL
GET
xMoverPathFree := THIS^._FB_ABL_100A.xOUT_MoverFree OR THIS^._FB_ABL_100A.xOUT_Ready OR THIS^._FB_ABL_100A.xOUT_Done;
END_GET
END_PROPERTY

PROPERTY xMoverShouldLeave : BOOL
GET
xMoverShouldLeave := THIS^._FB_ABL_100A.iOUT_Step = ST100_Load_e.SYNC_MOVER_LEAVE;
END_GET
END_PROPERTY

END_FUNCTION_BLOCK

// ---- POUs/20_AUTO/ST100/FB_AUT_UNLOAD.TcPOU
FUNCTION_BLOCK FB_AUT_UNLOAD EXTENDS FB_AUT_ABSTRACT IMPLEMENTS ISimuMoverTimers
(****************************************************************************)
(*	POU_AUT_zxx			Bausteinaufrufe Station	zxx							*)
(*	Status				ungetestet											*)
(*  Version:			1.0													*)
(*	Beschrieb:																*)
(*																			*)
(*	Abläufe:			FB_ABLzxxA		Hauptablauf							*)
(*																			*)
(*																			*)
(* 	25.09.2019/Dj															*)
(****************************************************************************)
(*	dd.mm.yyyy   KZ    x.y			Beschrieb								*)
(****************************************************************************)
VAR_INPUT
    (* spezifische Eingänge *)

END_VAR
VAR_OUTPUT
    (* spezifische Ausgänge *)

END_VAR
VAR
    (* Bausteine *)
    _FB_ABL_100A : FB_ABL_UNLOAD;
END_VAR

(*******************************************************************)
(* Timer *)
(*******************************************************************)

(*******************************************************************)
(* Flanken / Merker *)
(*******************************************************************)
//MANU CYCLE
IF (enIN_State = StateMANU) AND xIN_ManuCycle THEN
    xManuCycle := TRUE;
END_IF;

IF (enIN_State <> StateMANU) OR xOUT_Done THEN
    xManuCycle := FALSE;
END_IF

//NEXT STEP
xNextStep := (enIN_State > StateSTEP) OR
             ((enIN_State = StateSTEP) AND xIN_Step) OR
             ((enIN_State = StateMANU) AND xManuCycle);

//RESET
xReset := (enIN_State < StateREADY) AND (enIN_State <> StateINIT) AND NOT xManuCycle;

(*******************************************************************)
(* Bausteinaufrufe Abläufe *)
(*******************************************************************)

_FB_ABL_100A(xIN_Reset    := xReset,
             xIN_Init     := xIN_Init,
             xIN_Quit     := xIN_Quit,
             xIN_Start    := enIN_State = enState.StateAUTO, //AND _FB_ABL_100A.xOUT_Done AND _FB_ABL_100A.xOUT_Ready,
             xIN_Sperre   := NOT xIN_On,
             xIN_NextStep := xNextStep,
             xIN_AlarmAktiv
                 := xIN_AlarmAktiv,
             xIN_DryCycle    := xIN_DryCycle,
             xIN_RestartCYCL := enIN_State = enState.StateAUTO, // only restart when the mover has move out
             enIN_State      := enIN_State,
             tIN_Timeout     := tIN_Timeout,
             pxFG_Freigabe   := ADR(xRelease),
             Mover           := THIS^.Mover,
             xOUT_ErrFlag    =>,
             xOUT_Busy       =>,
             xOUT_Done       =>,
             xOUT_Timeout    =>,
             xOUT_InitDone   =>,
             xOUT_Wait       =>,
             iOUT_Step       =>,
             bOUT_Error      =>);

(*******************************************************************)
(* Mover reset flags *)
(*******************************************************************)

(*******************************************************************)
(* OUTPUT *)
(*******************************************************************)
xOUT_InitDone := _FB_ABL_100A.xOUT_InitDone;
xOUT_Ready    := xOUT_InitDone;
xOUT_Done     := _FB_ABL_100A.xOUT_Done;
xOUT_ErrFlag  := _FB_ABL_100A.xOUT_ErrFlag;
xOUT_Wait     := _FB_ABL_100A.xOUT_Wait;
xOUT_AlarmST  := xOUT_ErrFlag;

(*******************************************************************)
(* Bausteinaufruf Error Station *)
(*******************************************************************)
// POU_ERR_VORLAGE(xIN_QUIT:=xIN_Quit , pstrArIN_ALARM:=ADR(HMI.strArALARM[1]));

METHOD GiveMover : IProcessSampleMover
VAR_INPUT
	mover : REFERENCE TO FB_Mover;
END_VAR
IF __ISVALIDREF(mover) THEN
    THIS^.Mover REF= mover;
END_IF
END_METHOD

(* % of completion of the process *)
PROPERTY iCompletionPC : INT
GET
iCompletionPC := THIS^._FB_ABL_100A.iOUT_ProcessCompletion;
END_GET
END_PROPERTY

(* Process time, expressed in milisecond *)
PROPERTY iProcessTimeMili_1 : DINT
GET
iProcessTimeMili_1 := TO_DINT(this^._FB_ABL_100A.iProcessTimeMili1);
END_GET
SET
THIS^._FB_ABL_100A.iProcessTimeMili1 := TO_UDINT(iProcessTimeMili_1);
END_SET
END_PROPERTY

(* Process time, expressed in milisecond *)
PROPERTY iProcessTimeMili_2 : DINT
GET
iProcessTimeMili_2 := TO_DINT(this^._FB_ABL_100A.iProcessTimeMili2);
END_GET
SET
THIS^._FB_ABL_100A.iProcessTimeMili2 := TO_UDINT(iProcessTimeMili_2);
END_SET
END_PROPERTY

PROPERTY ProcessExecution : ProcessExecution_e
GET
ProcessExecution := THIS^._ProcessExecution;
END_GET
SET
THIS^._ProcessExecution := ProcessExecution;
END_SET
END_PROPERTY

METHOD TakeMover : IProcessSampleMover
VAR_INPUT
END_VAR
THIS^.Mover REF= 0;
END_METHOD

PROPERTY xBusy : BOOL
GET
xBusy := This^._FB_ABL_100A.xOUT_Busy;
END_GET
SET
END_SET
END_PROPERTY

PROPERTY xDone : BOOL
GET
xDone := THIS^._FB_ABL_100A.xOUT_Ready OR THIS^._FB_ABL_100A.xOUT_Done;
END_GET
END_PROPERTY

PROPERTY xMoverPathFree : BOOL
GET
xMoverPathFree := THIS^._FB_ABL_100A.xOUT_MoverFree OR THIS^._FB_ABL_100A.xOUT_Ready OR THIS^._FB_ABL_100A.xOUT_Done;
END_GET
END_PROPERTY

PROPERTY xMoverShouldLeave : BOOL
GET
xMoverShouldLeave := THIS^._FB_ABL_100A.iOUT_Step = ST100_Unload_e.SYNC_MOVER_LEAVE;
END_GET
END_PROPERTY

END_FUNCTION_BLOCK

// ---- POUs/20_AUTO/ST15x/FB_ABL_150_solo.TcPOU
FUNCTION_BLOCK FB_ABL_150_solo
(****************************************************************************************)
(*	TITEL				laden kristall- Modul	    										*)
(*	Status				ungetestet                         								*)
(*	Beschrieb:			Ablaufbeschreibung												*)
(*																						*)
(*	Steps:	self-explained using enum													*)
(***********************************Revisionen*******************************************)
(*	see github blames																	*)
(****************************************************************************************)

VAR_INPUT
    xIN_Reset       : BOOL;          // Schrittkette zurücksetzen 
    xIN_Init        : BOOL;          // Initialisieren
    xIN_Quit        : BOOL;          // Fehler quittieren 
    xIN_Start       : BOOL;          // Startbefehl
    xIN_Sperre      : BOOL;          // FB Sperren 
    xIN_NextStep    : BOOL;          // Nächsten Schritt ausführen 
    xIN_AlarmAktiv  : BOOL;          // Anlage hat Alarm
    xIN_DryCycle    : BOOL;          // Fahren ohne Teile
    xIN_RestartCYCL : BOOL;          // Zyklus erneut starten im STEP, END, LEERFAHREN
    enIN_State      : enState;       // Status Anlage
    tIN_Timeout     : TIME := T#10s; // Timout

    pxFG_Freigabe : POINTER TO BOOL; //Freigabe von Station

    // Application specific
    Mover : REFERENCE TO FB_Mover;

    xIN_capDetector             : BOOL;
    xIN_kraftubersetzunh_zuruck : BOOL;
    xIN_kraftubersetzunh_vor    : BOOL;

    xIN_welding_bits : Ultrasonic_IN_bits_t;

    iIN_StationNumber : INT; // station number 

END_VAR
VAR_OUTPUT
    (* standart Ausgänge *)
    xOUT_ErrFlag  : BOOL;        // Error Flag 
    xOUT_Busy     : BOOL;        // Baustein befindet sich im Ablauf 
    xOUT_Done     : BOOL;        // Baustein hat den Ablauf beendet 		
    xOUT_Ready    : BOOL;        // Ready to begin, should be the same state as done	
    xOUT_Timeout  : BOOL;        // Timeout FB 
    xOUT_InitDone : BOOL;        // initialisierung fertig
    xOUT_Wait     : BOOL;        // Wartet auf Bedingung
    iOUT_Step     : ST150_Uss_e; // Aktueller Schritt 
    sOUT_Step     : STRING;      // Aktueller Schritt but in string format
    bOUT_Error    : BYTE;        // Fehlernummer

    iOUT_ProcessCompletion : INT;  //process completion, express in % (0-100)
    xOUT_MoverFree         : BOOL; // The mover is free to move

    xOUT_moverMaintening_valve : BOOL;
    xOUT_welding_bits          : Ultrasonic_OUT_bits_t;

END_VAR
VAR
    (* Standard *)
    (* Schritt *)
    iLastStep : ST150_Uss_e; // Merker letzter Schritt 
    iPreStep  : ST150_Uss_e; // Schritt zurück nach Alarm 
    iAktStep  : ST150_Uss_e; // aktueller Schritt

    // Trigger Starten 
    rtSTART : R_TRIG;
    // Timer TimeOut 
    TON_Timeout : TON;

    (* Bausteine *)

    (* Spezial *)
    fb_moverMaintening   : FB_ZylMo2El_V2_1;
    simu_moverMaintening : FB_Simu_Zyl2Pos;

    TON_UssError : TON;

    welding_right_done    : BOOL := FALSE;
    ton_wait_mover_in_pos : TON;

END_VAR
VAR CONSTANT
    USS_SIMULATION : BOOL := FALSE; // Set to TRUE to simulate this part of the program
END_VAR

(*******************************************************************)
(* Trigger  *)
(*******************************************************************)
(* Zurücksetzen *)
IF xIN_RESET THEN
    iPreStep  := ST150_Uss_e.RESET;
    iOUT_Step := ST150_Uss_e.RESET;
END_IF;

(* Error Quittieren *)
IF (bOUT_Error <> 0) AND xIN_Quit THEN
    xOUT_ErrFlag := FALSE;
    bOUT_Error   := 0;
    iOUT_Step    := ST150_Uss_e.INIT;
END_IF;

(*******************************************************************)
(* Timer *)
(*******************************************************************)
TON_Timeout(IN := xIN_NextStep AND (iLastStep = iOUT_Step) (*todo FG *) ,
            PT := tIN_Timeout);

TON_UssError(IN := ST150_Uss_e.uss_start = iOUT_Step,
             PT := DINT_TO_TIME(_20_AUTO.recipe.st150.USS_ErrorTime_ms));

ton_wait_mover_in_pos(IN := iOUT_Step = ST150_Uss_e.wait_shuttle_in_pos,
                      PT := T#1S);

(*******************************************************************)
(* Bausteine *)
(*******************************************************************)
fb_moverMaintening(xIN_Reset    := xIN_Reset OR (ST150_Uss_e.RESET = iOUT_Step),
                   xIN_Quit     := xIN_Quit,
                   xIN_Manu     := enState.StateMANU = enIN_State,
                   pbtIN_Button := ADR(HMI.btManuCylinders[StationList_e.ST150][1]),
                   xIN_GS       := simu_moverMaintening.xOUT_inGS,
                   xIN_AS       := simu_moverMaintening.xOUT_inAS,
                   xIN_FREE     := TRUE,
                   xINtoGS      := (ST150_Uss_e.Init_ResetUss_maintaining_down = iOUT_Step) OR
                                   (ST150_Uss_e.mover_maintening_down = iOUT_Step),
                   xINtoAS   := ST150_Uss_e.mover_maintening_up = iOUT_Step,
                   tIN_ErrAS := DINT_TO_TIME(_20_AUTO.recipe.cylinder2Pos[StationList_e.ST150]
                                                 [ST150_Cylinders_e.Kraftbstutzung].toAS_alarm_time),
                   tIN_ErrGS := DINT_TO_TIME(_20_AUTO.recipe.cylinder2Pos[StationList_e.ST150]
                                                 [ST150_Cylinders_e.Kraftbstutzung].toGS_alarm_time),
                   tIN_WaitAS := DINT_TO_TIME(_20_AUTO.recipe.cylinder2Pos[StationList_e.ST150]
                                                  [ST150_Cylinders_e.Kraftbstutzung].toAS_wait_time),
                   tIN_WaitGS := DINT_TO_TIME(_20_AUTO.recipe.cylinder2Pos[StationList_e.ST150]
                                                  [ST150_Cylinders_e.Kraftbstutzung].toGS_wait_time));

simu_moverMaintening(xIN_Enable := USS_SIMULATION AND CONST.USE_SIMULATION,
                     xIN_inGS   := xIN_kraftubersetzunh_zuruck,
                     xIN_inAS   := xIN_kraftubersetzunh_vor,
                     xIN_valve  := fb_moverMaintening.xOUT_VALVE,
                     tIN_GS_ms  := 200,  // ms
                     tIN_AS_ms  := 200); // ms

(*******************************************************************)
(* OUTPUTS *)
(*******************************************************************)
// Error Flag 
xOUT_ErrFlag := (bOUT_Error <> 0) OR (ST150_Uss_e.ERROR = iOUT_Step);
// Baustein befindet sich im Ablauf 
xOUT_Busy := (iOUT_Step > ST150_Uss_e.READY) AND (iOUT_Step < ST150_Uss_e.DONE);
// Baustein hat den Ablauf beendet
xOUT_Done := (iOUT_Step = ST150_Uss_e.DONE);
// Process ready
xOUT_Ready := (iOUT_Step = ST150_Uss_e.READY) OR (iOUT_Step = ST150_Uss_e.waitOnMover);
// Timeout FB 				 		
xOUT_Timeout := TON_Timeout.Q;
// Itialisierung fertig			
xOUT_InitDone := (iOUT_Step = ST150_Uss_e.READY) OR (iOUT_Step = ST150_Uss_e.waitOnMover);
// Aktueller Schritt			
iOUT_Step := iOUT_Step; //Im Ablauf gesetzt		
sOUT_Step := TO_STRING(iOUT_Step);
//Fehlernummer	 
bOUT_Error := bOUT_Error; //Im Ablauf/FB gesetzt	
(* Warte (alle Schritte wo auf FG oder Teile gewartet wird) *)
xOUT_Wait := (iOUT_Step = ST150_Uss_e.DONE) OR
             (iOUT_Step = ST150_Uss_e.READY) OR
             (iOUT_Step = ST150_Uss_e.START) OR
             (iOUT_Step = ST150_Uss_e.waitOnMover) OR
             (iOUT_Step = ST150_Uss_e.SYNC_MOVER_LEAVE);

xOUT_MoverFree := iOUT_Step >= ST150_Uss_e.MOVER_FREE_OP AND iOUT_Step < ST150_Uss_e.MOVER_NEEDED_OP;

iOUT_ProcessCompletion := F_GetPercent_2(iAktStep,
                                         iAktStep,
                                         iAktStep,
                                         ST150_Uss_e.check_cap_present,
                                         ST150_Uss_e.SYNC_MOVER_LEAVE);

xOUT_moverMaintening_valve :=
    fb_moverMaintening.xOUT_VALVE AND NOT (USS_SIMULATION AND CONST.USE_SIMULATION);

xOUT_welding_bits.Start :=
    (ST150_Uss_e.uss_start = iOUT_Step) AND
    NOT (USS_SIMULATION AND CONST.USE_SIMULATION) AND
    xIN_capDetector;

xOUT_welding_bits.Reset :=
    _14_STATE._FB_btQUIT.pbtIN^.press OR (ST150_Uss_e.Init_ResetUss_maintaining_down = iOUT_Step);

xOUT_welding_bits.Data_Hex1 := _20_AUTO.recipe.st150.USS_Type.0; // _20_AUTO.recipe.st150.USS_Type = 1;
xOUT_welding_bits.Data_Hex2 := _20_AUTO.recipe.st150.USS_Type.1; // _20_AUTO.recipe.st150.USS_Type = 2;
xOUT_welding_bits.Data_Hex4 := _20_AUTO.recipe.st150.USS_Type.2; // _20_AUTO.recipe.st150.USS_Type = 3;
xOUT_welding_bits.Data_Hex8 := _20_AUTO.recipe.st150.USS_Type.3; // _20_AUTO.recipe.st150.USS_Type = 4;

(*******************************************************************)
(* Ablauf *)
(*******************************************************************)

(* Sperren *)
IF xIN_Sperre THEN
    iPreStep  := ST150_Uss_e.RESET;
    iOUT_Step := ST150_Uss_e.RESET;
    RETURN;
END_IF;

(* Schritt Merker *)
IF iAktStep <> iOUT_Step THEN
    iLastStep := iAktStep;
    iAktStep  := iOUT_Step;
END_IF

(* START *)
rtSTART(CLK := xIN_Start);

IF 0 = bOUT_Error THEN
    IF fb_moverMaintening.xOUT_ErrFlag THEN
        bOUT_Error := 11;
    ELSIF USS_SIMULATION AND CONST.USE_SIMULATION AND xIN_welding_bits.Fehler THEN
        bOUT_Error := 12;
    ELSIF TON_UssError.Q THEN
        bOUT_Error := 13;
    END_IF
ELSIF iOUT_Step < ST150_Uss_e.ERROR THEN
    iOUT_Step := ST150_Uss_e.ERROR;
END_IF

(*******************************************************************)
(* Schrittkette  *)
(*******************************************************************)
CASE iOUT_Step OF

(***** RESET *****)
ST150_Uss_e.RESET: (* Schritt 0-99 *)
    //Initialisierungen
    //Start Init Ablauf
    IF xIN_Init THEN
        iOUT_Step := ST150_Uss_e.INIT;
        //Start Manu Ablauf
    ELSIF enIN_State = StateMANU AND xIN_NextStep THEN
        iOUT_Step := ST150_Uss_e.INIT;
    END_IF;

(***** INIT *****)
ST150_Uss_e.INIT: (* Grundstellung ? *)
    iOUT_Step := ST150_Uss_e.Init_ResetUss_maintaining_down;

ST150_Uss_e.Init_ResetUss_maintaining_down:
    IF fb_moverMaintening.xOUT_inGS THEN
        iOUT_Step := ST150_Uss_e.READY;
    END_IF

(***** READY / INIT DONE *****)
ST150_Uss_e.READY:    (* Start AUTO,END,LEER,STEP *)
    IF xIN_Start THEN //IF rtSTART.Q THEN
        iOUT_Step := ST150_Uss_e.START;
    END_IF

(***** START  ZYKLISCH *****)
ST150_Uss_e.START: (*  *)
    IF xIN_NextStep AND pxFG_Freigabe^ THEN
        iOUT_Step := ST150_Uss_e.waitOnMover;
    END_IF;

ST150_Uss_e.waitOnMover: (*  *)
    IF xIN_NextStep AND __ISVALIDREF(Mover) THEN
        IF Mover.GetLastStationDone() >= iIN_StationNumber THEN
            iOUT_Step := ST150_Uss_e.SYNC_MOVER_LEAVE;
        ELSE
            iOUT_Step := ST150_Uss_e.mover_maintening_up;
        END_IF
    END_IF;

ST150_Uss_e.check_cap_present:
    IF xIN_capDetector OR (USS_SIMULATION AND CONST.USE_SIMULATION) THEN
        iOUT_Step := ST150_Uss_e.mover_maintening_up;
    ELSE
        iOUT_Step := ST150_Uss_e.SYNC_MOVER_LEAVE;

        IF __ISVALIDREF(Mover) THEN
            IF NOT Mover.SetLastStation(-iIN_StationNumber) THEN
                ASSERT(0);
            END_IF
        END_IF
    END_IF

ST150_Uss_e.mover_maintening_up:
    IF xIN_NextStep AND fb_moverMaintening.xOUT_inAS THEN
        IF USS_SIMULATION AND CONST.USE_SIMULATION THEN
            iOUT_Step := ST150_Uss_e.mover_maintening_down;
        ELSE
            IF xIN_welding_bits.Bereit THEN
                iOUT_Step := ST150_Uss_e.uss_start;

                IF __ISVALIDREF(Mover) THEN
                    IF NOT Mover.SetLastStation(-150) THEN
                        ASSERT(0);
                    END_IF
                END_IF
            ELSE
                bOUT_Error := 1; // welding not ready
            END_IF
        END_IF;
    END_IF;

ST150_Uss_e.uss_start:
    IF xIN_NextStep AND NOT xIN_welding_bits.NullPosition THEN
        iOUT_Step := ST150_Uss_e.uss_working;
    END_IF

ST150_Uss_e.uss_working:
    IF xIN_NextStep AND
       (NOT xIN_welding_bits.US_on AND
       xIN_welding_bits.NullPosition) THEN
        iOUT_Step := ST150_Uss_e.mover_maintening_down;
    END_IF

ST150_Uss_e.mover_maintening_down:
    IF xIN_NextStep AND fb_moverMaintening.xOUT_inGS THEN
        iOUT_Step := ST150_Uss_e.move_shuttle_120_mm;
    END_IF;

ST150_Uss_e.move_shuttle_120_mm:
    IF xIN_NextStep AND __ISVALIDREF(Mover) AND_THEN Mover.MoveRelativeInsideStation(118.0) THEN
        iOUT_Step := ST150_Uss_e.wait_shuttle_in_pos;
    END_IF

ST150_Uss_e.wait_shuttle_in_pos:
    IF ton_wait_mover_in_pos.Q THEN
        IF welding_right_done THEN
            iOUT_Step          := ST150_Uss_e.SYNC_MOVER_LEAVE;
            welding_right_done := FALSE;

            IF __ISVALIDREF(Mover) THEN
                IF NOT Mover.SetLastStation(iIN_StationNumber) THEN
                    ASSERT(0);
                END_IF
            END_IF
        ELSE
            iOUT_Step          := ST150_Uss_e.check_cap_present;
            welding_right_done := TRUE;
        END_IF
    END_IF

ST150_Uss_e.SYNC_MOVER_LEAVE:
    // The mover needs to be taken by MoverMan
    IF NOT __ISVALIDREF(Mover) THEN
        iOUT_Step := ST150_Uss_e.DONE;
    END_IF

(***** DONE *****)
ST150_Uss_e.DONE: (* Letzter Schritt  *)
    IF NOT xIN_AlarmAktiv THEN
        //AUTO
        IF (enIN_State = StateAUTO) AND xIN_RestartCYCL THEN
            iOUT_Step := ST150_Uss_e.START;
            //STEP / END / LEERFAHREN restart
        ELSIF (enIN_State < StateAUTO) AND (enIN_State >= enState.StateSTEP) AND xIN_RestartCYCL THEN
            iOUT_Step := ST150_Uss_e.START;
            //STEP / END / LEERFAHREN fertig
        ELSIF (enIN_State = StateREADY) THEN
            iOUT_Step := ST150_Uss_e.READY;
        END_IF;
    END_IF;

(************ ERROR *************)
ST150_Uss_e.ERROR: (* ERROR *) ;

END_CASE;

END_FUNCTION_BLOCK

// ---- POUs/20_AUTO/ST175/Trumpf/TruMark_Ethercat_dj.TcPOU
PROGRAM TruMark_Ethercat_dj
VAR
    // EtherCat Zustand
    uiECatStatus AT %I* : UINT; // --> Status von ECAT-Klemme (101A2-InfoData-State)
    wStateMachine       : WORD;

    // Bus-Structure - Input
    PBIM0 AT %I* : ARRAY[0..1] OF WORD;  // --> Linked with EK1110. TxPDO. Byte 0 - 3
    PBIM1 AT %I* : ARRAY[0..1] OF WORD;  // --> Linked with EK1110. TxPDO. Byte 4 - 7
    PBIM2 AT %I* : ARRAY[0..63] OF WORD; // --> Linked with EK1110. TxPDO. Byte 8 - 135

    // Bus-Structure - Output
    PBOM0 AT %Q* : ARRAY[0..1] OF WORD;  // --> Linked with EK1110. RxPDO. Byte 0 - 3
    PBOM1 AT %Q* : ARRAY[0..1] OF WORD;  // --> Linked with EK1110. RxPDO. Byte 3 - 7
    PBOM2 AT %Q* : ARRAY[0..63] OF WORD; // --> Linked with EK1110. RxPDO. Byte 8 - 135

    // TLV Data Structure
    awTlvPBxM2 : if_Command_u;

    // BIT Helper-Variables
    // awPBOM AT %M* : ARRAY[0..1] OF WORD;
    // dwPBOM AT %M* : DWORD;

    iStep    : INT;
    t1       : TON;
    bT1Start : BOOL;
    sS1      : STRING;
    iInd     : INT;
END_VAR

t1(IN := bT1Start, PT := T#2000MS);
wStateMachine := UINT_TO_WORD(uiECatStatus) AND 16#00FF;

IF wStateMachine <> 8 THEN
    if_TruMark.bError := TRUE;
    iStep             := 0;
END_IF

IF (iStep = 99) AND HMI.btArMain[7].rtrig THEN
    if_TruMark.bResetErr := TRUE;
END_IF

if_TruMark.Status.b0_Laser_On                  := PBIM0[0].0;
if_TruMark.Status.b1_Laser_Ready               := PBIM0[0].1;
if_TruMark.Status.b2_SIK_Open                  := PBIM0[0].2;
if_TruMark.Status.b3_Shutter_Open              := PBIM0[0].3;
if_TruMark.Status.b4_BeamExpander_IsInPos      := PBIM0[0].4;
if_TruMark.Status.b5_LaserMonitoring           := PBIM0[0].5;
if_TruMark.Status.b6_LaserMalfunction          := PBIM0[0].6;
if_TruMark.Status.b7_PilotLaser_On             := PBIM0[0].7;
if_TruMark.Status.b8_LaserWarningLamp_On       := PBIM0[0].8;
if_TruMark.Status.b9_QSwTrigger_ON             := PBIM0[0].9;
if_TruMark.Status.b10_SwOff_NotActivated       := PBIM0[0].10;
if_TruMark.Status.b11_KeySwLaserDisable_Closed := PBIM0[0].11;
if_TruMark.Status.b12_EmergencyStop_Closed     := PBIM0[0].12;
if_TruMark.Status.b13_LaserHeatingPhase_On     := PBIM0[0].13;
if_TruMark.Status.b14_ControlUnit_On           := PBIM0[0].14;
if_TruMark.Status.b15_Mark_Active              := PBIM0[0].15;
if_TruMark.Status.b16_Conversion_Active        := PBIM0[1].0;

CASE iStep OF
0: // Bus Initialisation
    CASE wStateMachine OF
    8: // 'OP';
        if_TruMark.sErrorMsg := '';
        if_TruMark.bError    := FALSE;
        if_TruMark.bBusy     := FALSE;
        if_TruMark.bBitCmd   := FALSE;
        if_TruMark.bTlvCmd   := FALSE;
        if_TruMark.bResetErr := FALSE;
        iStep                := 5;
    ELSE
        if_TruMark.sErrorMsg :=
            CONCAT('EtherCat Bus ist nicht bereit.  State Machine = ', UINT_TO_STRING(wStateMachine));
    END_CASE

5: // Waiting for command (TLV or BIT)
    IF if_TruMark.bBitCmd THEN
        if_TruMark.bBusy := TRUE;
        iStep            := 10;
    END_IF

    IF if_TruMark.bTlvCmd THEN
        if_TruMark.bBusy           := TRUE;
        if_TruMark.byTlvExtErrCode := 0;
        if_TruMark.byTlvReturnCode := 0;
        iStep                      := 20;
    END_IF

10: // ------------------------------------
    // BIT Command
    // ------------------------------------
    awTlvPBxM2.as_struct.bit_command.dwPBOM := if_TruMark.dwBitIn;
    PBOM0                                   := awTlvPBxM2.as_struct.bit_command.awPBOM;
    iStep                                   := 0;

20: // ------------------------------------
    // TLV Command
    // ------------------------------------
    awTlvPBxM2.as_struct.diTlvTag := if_TruMark.diTlvTag;

    // Convert String to ASCII Code
    FOR iInd := 0 TO LEN(if_TruMark.sTlvValueIn) BY 1 DO
        IF if_TruMark.sTlvValueIn[iInd] = 16#3B THEN
            awTlvPBxM2.as_struct.abyTlvValues[iInd] := 16#00;
        ELSE
            awTlvPBxM2.as_struct.abyTlvValues[iInd] := if_TruMark.sTlvValueIn[iInd];
        END_IF
    END_FOR

    awTlvPBxM2.as_struct.abyTlvValues[iInd] := 16#00;
    awTlvPBxM2.as_struct.diTlvLenght        := INT_TO_DINT(iInd);

    // 1.   A T T E N T I O N  - copy first all Data on the bus
    PBOM2 := awTlvPBxM2.as_word_array;

    // 2.   A T T E N T I O N  - then set a new Handshake --> a new Handshake will trigger a command
    PBOM2[0] := PBIM2[0] + 1; // increment Handshake

    IF PBOM2[0] < 2 OR PBOM2[0] > 255 THEN // Valid Range for Handshake is between 2 and 255
        PBOM2[0] := 2;                     // minimal Handshake
    END_IF

    iStep := 21;

21: // Waiting for TLV-Response
    // A TLV-Response has a new handshake (newHS = oldHS + 1)
    // The response time varries depending on the TLV request/command
    IF PBOM2[0] <= PBIM2[0] THEN
        awTlvPBxM2.as_word_array   := PBIM2;
        if_TruMark.byTlvReturnCode := awTlvPBxM2.as_struct.abyTlvValues[0];

        CASE if_TruMark.byTlvReturnCode OF
        16#30: // Ascii = '0'		- No Error
            sS1 := '';

            FOR iInd := 0 TO DINT_TO_INT(awTlvPBxM2.as_struct.diTlvLenght - 1) BY 1 DO
                IF awTlvPBxM2.as_struct.abyTlvValues[iInd] = 16#00 THEN
                    sS1 := CONCAT(STR1 := sS1, STR2 := ';');
                ELSE
                    sS1 := CONCAT(STR1 := sS1, STR2 := F_ToCHR(c := awTlvPBxM2.as_struct.abyTlvValues[iInd]));
                END_IF
            END_FOR

            if_TruMark.sTlvRespons := sS1;
            iStep                  := 0;

        16#31: // Ascii = '1'
            if_TruMark.bError          := TRUE;
            if_TruMark.sErrorMsg       := 'TLV Error: Command was not executed!';
            if_TruMark.byTlvExtErrCode := awTlvPBxM2.as_struct.abyTlvValues[2];
            iStep                      := 99;

        16#32: // Ascii = '2'
            if_TruMark.bError    := TRUE;
            if_TruMark.sErrorMsg := 'TLV Error: Invalid parameter value!';
            iStep                := 99;

        16#33: // Ascii = '3'
            if_TruMark.bError    := TRUE;
            if_TruMark.sErrorMsg := 'TLV Error: Invalid TLV value lenght!';
            iStep                := 99;
        ELSE
            if_TruMark.bError    := TRUE;
            if_TruMark.sErrorMsg := 'TLV Error';
            iStep                := 99;
        END_CASE
    END_IF

99: // in case of an TLV Error
    if_TruMark.bBusy := FALSE;

    IF if_TruMark.bResetErr THEN
        iStep := 0;
    END_IF

END_CASE

END_PROGRAM

// ---- GlobalTextList.TcGTLO
TEXTLIST GlobalTextList
  372 = ' Integral-action time [ms] Tn'
  1330 = ' Integral-action time [s]'
  742 = ' Integral-action time [s] Tn'
  767 = '$'
  18 = '%.2f'
  1316 = '%.3f'
  1260 = '%.d'
  1413 = '%1.3f'
  373 = '%d'
  962 = '%f'
  999 = '%s'
  1561 = '1 = Maxi     2 = Pro    3 = Smart & Mini'
  148 = '30000'
  193 = 'Accel Override'
  283 = 'Acceleration'
  166 = 'Acceleration:'
  1776 = 'All ids set'
  1495 = 'at target'
  632 = 'AUTO'
  1133 = 'Available type :\n30L : 1'
  398 = 'Available type :\nJURA 50l : 1'
  364 = 'Available type :\nJURA 50l = 1'
  2269 = 'Available type :\nJURA 50l = 1\nJURA 120l = 2\nJURA 30l = 3\nFreezio 120l = 1\nDaempfer 130l = 1'
  827 = 'Available type :\nJURA 50l = 1\nJURA 120l = 2\nJURA 30l = 3\nFreezio 120l = 1\nDaempfer 130l = 1\nDaempfer 130l = 1'
  2185 = 'Available type :\nJURA 50l = 1\nJURA 120l = 2\nJURA 30l = 3\nFreezio 120l = 1\nDaempfer 130l = 1\nJURA 300l = 1'
  1753 = 'Available type :\nJURA 50l = 1\nJURA 120l = 2\nJURA 30l = 3\nFreezio 120l = 1\nJURA 50l = 1'
  2163 = 'Available type :\nJURA 50l = 1\nJURA 120l = 2\nJURA 30l = 3\nFreezio 120l = 4\nDaempfer 130l = 5\nJURA 300l = 6'
  1533 = 'Available type :\nJURA 50l = 1\nJURA 50l = 1\nJURA 50l = 1\nJURA 50l = 1\nJURA 50l = 1'
  1504 = 'Available type :\nJURA 50l, Type 1 : 1'
  1745 = 'Available type :\nSMART_MINI\nSMART\nBLUE\nSMART_KRISTALL\nBLUE_KRISTALL\nPRO_SMART\nPRO_BLUE\nPRO_SMART_KRISTALL\nPRO_SMART_MAXI\nPRO_SMART_MAXI_KRISTALL'
  34 = 'Available type :SMART_MINI\nSMART\nBLUE\nSMART_KRISTALL\nBLUE_KRISTALL\nPRO_SMART\nPRO_BLUE\nPRO_SMART_KRISTALL\nPRO_SMART_MAXI\nPRO_SMART_MAXI_KRISTALL'
  404 = 'Avg'
  380 = 'Copy'
  758 = 'Copy default'
  223 = 'Copy recipe to:'
  460 = 'current'
  209 = 'Current height sensor value'
  998 = 'Current state:'
  51 = 'Cylinder config'
  491 = 'Cylinder list:'
  729 = 'Damping time [ms] Td'
  454 = 'Damping time [s] Td'
  453 = 'Decel Override'
  1020 = 'Deceleration'
  36 = 'Default value :'
  1832 = 'Derivative action time [ms] Tv'
  170 = 'Derivative action time [s] Tv'
  726 = 'Done to Done'
  2481 = 'Done to Done : '
  802 = 'EmptyDelay'
  500 = 'Enable power'
  1713 = 'Enable process'
  1317 = 'Enable RUN'
  423 = 'Enable SuperTrak'
  921 = 'enablePower'
  203 = 'END'
  165 = 'error'
  1052 = 'error :'
  1880 = 'error:'
  1329 = 'farward dir'
  1402 = 'Farward direction'
  919 = 'FeederConfig Left'
  241 = 'FeederConfig Right'
  986 = 'FeederConfig.EmptyDelay'
  446 = 'FeederConfig.InFilterDelay'
  1207 = 'FeederConfig.StartDelay'
  1185 = 'FeederConfig.StopDelay'
  938 = 'Fifo len = %d'
  642 = 'File name (no extension, no path)'
  347 = 'Force'
  1236 = 'Force is in place'
  1049 = 'Force place'
  28 = 'in operation'
  354 = 'in position'
  976 = 'InFilterDelay'
  557 = 'INIT'
  341 = 'Is type smart or mini ?'
  1715 = 'Is X offset negative'
  1617 = 'Is Y offset negative'
  275 = 'Is Z height negative'
  93 = 'Jerk'
  688 = 'Jerk Override'
  41 = 'kraft sensor detect left'
  1013 = 'kraft sensor detect right'
  587 = 'kraft sensor limit left'
  820 = 'LEER'
  49 = 'Linear Axis'
  1256 = 'Load kammer'
  779 = 'Load kammer time [ms]'
  485 = 'Load mixture time'
  1289 = 'Load Patrone time [ms]'
  561 = 'lost pos feedback'
  905 = 'MANU'
  641 = 'Max'
  1293 = 'max height'
  1284 = 'max height left'
  1994 = 'max height left or middle'
  717 = 'max height right'
  23 = 'Max speed:'
  386 = 'Min'
  1167 = 'min height'
  975 = 'min height left'
  579 = 'min height left or middle'
  1588 = 'min height right'
  615 = 'Move farward'
  407 = 'Move farward direction'
  426 = 'Move list :'
  238 = 'Move reverse direction'
  33 = 'Move without movers / WF'
  716 = 'Mover 1 actual pos :'
  50 = 'Mover details'
  357 = 'Mover n°'
  48 = 'Mover Track'
  826 = 'moving farward'
  1573 = 'moving reverse'
  192 = 'moving to target'
  1333 = 'Next station :'
  103 = 'Offset'
  583 = 'Piece good max height'
  908 = 'Piece good min height'
  375 = 'Piece holder:'
  251 = 'Position'
  1318 = 'power on'
  639 = 'Process name:'
  2584 = 'Program number'
  520 = 'Program number ST160'
  1188 = 'Program number ST165'
  1143 = 'Proportional amplification Kp'
  566 = 'QUIT'
  63 = 'ready'
  1608 = 'recovering'
  1477 = 'RELEASE'
  1460 = 'release unknown shuttle'
  1483 = 'Reset errors'
  299 = 'RESET POWER'
  849 = 'RESET TEMP COUNTER'
  556 = 'resetErrors'
  94 = 'reverse dir'
  1084 = 'Reverse direction'
  1168 = 'RFID Type'
  1593 = 'Robo'
  977 = 'Robot'
  2678 = 'Rotary table offset [°]'
  2718 = 'Running time :'
  832 = 'Save var'
  990 = 'Select axis :'
  1472 = 'Select recipe:'
  358 = 'servo_enabled'
  105 = 'SET'
  630 = 'Set all mover ApproachScenario'
  84 = 'Set all station time'
  421 = 'Set default'
  523 = 'set shuttle number'
  11 = 'Shuttle to unload'
  1396 = 'Shuttles to unload'
  1914 = 'Slot number of the rotary table'
  2049 = 'Smart or smart mini ?'
  1062 = 'SMART_MINI\nSMART\nBLUE\nSMART_KRISTALL\nBLUE_KRISTALL\nPRO_SMART\nPRO_BLUE\nPRO_SMART_KRISTALL\nPRO_SMART_MAXI\nPRO_SMART_MAXI_KRISTALL'
  1759 = 'ST 105'
  361 = 'ST 110'
  842 = 'ST 115'
  152 = 'ST 120'
  234 = 'ST 125'
  685 = 'ST 130'
  1076 = 'ST 145'
  560 = 'ST 160 Use left element'
  771 = 'ST 180'
  280 = 'ST 185'
  367 = 'ST105'
  52 = 'ST105 - Feeder'
  2158 = 'ST105 - Pnp'
  1614 = 'ST105 Configuration'
  965 = 'ST110'
  605 = 'ST110 - Feeder'
  2317 = 'ST110 - Pnp'
  248 = 'ST110 Configuration'
  902 = 'ST115'
  1777 = 'ST115 - Feeder'
  1136 = 'ST115 Configuration'
  633 = 'ST120'
  837 = 'ST120 - Feeder'
  1099 = 'ST120 Configuration'
  304 = 'ST125'
  2314 = 'ST125 - Feeder'
  840 = 'ST125 Configuration'
  810 = 'ST128'
  610 = 'ST130'
  1895 = 'ST130 - Dosieren'
  173 = 'ST130 Configuration'
  108 = 'ST135'
  53 = 'ST135 - Dosieren'
  328 = 'ST140'
  2618 = 'ST140 - Measure'
  578 = 'ST140 Configuration'
  559 = 'ST145'
  2143 = 'ST145 - Feeder'
  31 = 'ST145 Configuration'
  406 = 'ST150'
  703 = 'ST150 - Uss'
  167 = 'ST150 / 155 Configuration'
  509 = 'ST150 Configuration'
  30 = 'ST155'
  1199 = 'ST155 - Uss'
  326 = 'ST160'
  2461 = 'ST160 - CETA'
  1611 = 'ST160 / 165 Configuration'
  1826 = 'ST160 Use left element'
  2265 = 'ST160 Use right element'
  841 = 'ST165'
  1863 = 'ST165 - CETA'
  607 = 'ST165 Use left element'
  1110 = 'ST165 Use right element'
  619 = 'ST170'
  1873 = 'ST170 - RFID'
  1906 = 'ST170 Configuration'
  1379 = 'ST170 Use left element'
  1075 = 'ST170 Use right element'
  1638 = 'ST174'
  492 = 'ST175'
  199 = 'ST175 - LASER'
  2195 = 'ST175 Configuration'
  422 = 'ST176'
  415 = 'ST180'
  322 = 'ST180 Configuration'
  710 = 'ST185'
  1258 = 'start numbering sequence'
  493 = 'StartDelay'
  1283 = 'startMoverNumberingSequence'
  1322 = 'Station'
  702 = 'Station name:'
  645 = 'STEP'
  457 = 'STOP'
  325 = 'Stop mover'
  1080 = 'StopDelay'
  1178 = 'Timing'
  577 = 'toAS_alarm_time'
  397 = 'toAS_wait_time'
  194 = 'TOF blow element'
  1639 = 'toGS_alarm_time'
  1135 = 'toGS_wait_time'
  157 = 'TON sensor tube presence left'
  878 = 'TON sensor tube presence right'
  187 = 'TON wait time before blow'
  741 = 'TON_WaitPieceTime'
  847 = 'Trigger Pos'
  627 = 'Trigger Type'
  317 = 'Trigger Type:     0 = n.a.   1=SetPos    2=FromLast    3=FromEnd'
  239 = 'Use left element'
  1 = 'Use right element'
  769 = 'Use vertical left element'
  1275 = 'Use vertical right element'
  39 = 'USS Bereit'
  181 = 'USS Fehler'
  408 = 'USS null pos'
  876 = 'USS Reset'
  385 = 'USS reset'
  410 = 'USS Start'
  567 = 'USS start'
  2459 = 'Uss timeout [ms]'
  2030 = 'Uss Type'
  447 = 'USS us on'
  506 = 'Vacum treshold left [%]'
  679 = 'Vacum treshold right [%]'
  712 = 'Velo Override'
  879 = 'Velocity (0-100%)'
  371 = 'Vereinzelung piece bad max height'
  82 = 'Vereinzelung piece bad min height'
  588 = 'Vereinzelung Piece good max height'
  954 = 'Vereinzelung piece good max height'
  1208 = 'Vereinzelung piece good min height'
  487 = 'Vibration force underneath  [ms]'
  808 = 'Vibration force underneath [%]'
  339 = 'View 105'
  10 = 'View 110'
  896 = 'View 115'
  55 = 'View 120'
  301 = 'View 125'
  1925 = 'View 128'
  593 = 'View 130'
  1328 = 'View 140'
  1078 = 'View 145'
  1887 = 'View 15x'
  558 = 'View 16x'
  2155 = 'View 170'
  2495 = 'View 175'
  290 = 'View 180'
  656 = 'View 185'
  723 = 'Waiting time :'
  1793 = 'Whole path free'
  1691 = 'with offset :'
  1702 = 'with offset [um] :'
  1624 = 'X offset for pick position'
  1581 = 'X offset for pick position [0.1 mm]'
  1074 = 'Y offset for pick position [0.1 mm]'
  1899 = 'Y offset of the piece'
  1716 = 'Y offset of the piece [0.1 mm]'
  424 = 'Y offset of the piece [0.1mm]'
  1684 = 'Y offset of thepiece'
  1635 = 'Z height of the piece'
  1900 = 'Z height of the piece [0.1 mm]'
  242 = '[ms]'
END_TEXTLIST

